LIN {X 0,Y 213.972,Z 422.456,A -85,B 0,C 180,E1 -20686.708,E2 -20686.708} C_VEL
LIN {X 0,Y 214.158,Z 422.425,A -85,B 0,C 180,E1 -20690.556,E2 -20690.556} C_VEL
LIN {X 0,Y 214.219,Z 422.426,A -85,B 0,C 180,E1 -20692.46,E2 -20692.46} C_VEL
LIN {X 0,Y 214.439,Z 422.398,A -85,B 0,C 180,E1 -20698.122,E2 -20698.122} C_VEL
LIN {X 0,Y 214.546,Z 422.38,A -85,B 0,C 180,E1 -20700,E2 -20700} C_VEL
LIN {X 0,Y 214.44,Z 422.395,A -85,B 0,C 180,E1 -20701.879,E2 -20701.879} C_VEL
LIN {X 0,Y 214.219,Z 422.4,A -85,B 0,C 180,E1 -20707.541,E2 -20707.541} C_VEL
LIN {X 0,Y 214.037,Z 422.432,A -85,B 0,C 180,E1 -20711.363,E2 -20711.363} C_VEL
LIN {X 0,Y 213.926,Z 422.461,A -85,B 0,C 180,E1 -20715.238,E2 -20715.238} C_VEL
LIN {X 0,Y 213.832,Z 422.475,A -85,B 0,C 180,E1 -20719.189,E2 -20719.189} C_VEL
LIN {X 0,Y 213.84,Z 422.469,A -85,B 0,C 180,E1 -20723.228,E2 -20723.228} C_VEL
LIN {X 0,Y 213.822,Z 422.463,A -85,B 0,C 180,E1 -20727.451,E2 -20727.451} C_VEL
LIN {X 0,Y 213.761,Z 422.467,A -85,B 0,C 180,E1 -20731.739,E2 -20731.739} C_VEL
LIN {X 0,Y 213.738,Z 422.473,A -85,B 0,C 180,E1 -20736.29,E2 -20736.29} C_VEL
LIN {X 0,Y 213.708,Z 422.488,A -85,B 0,C 180,E1 -20741.127,E2 -20741.127} C_VEL
LIN {X 0,Y 213.772,Z 422.468,A -85,B 0,C 180,E1 -20746.342,E2 -20746.342} C_VEL
LIN {X 0,Y 213.734,Z 422.475,A -85,B 0,C 180,E1 -20751.339,E2 -20751.339} C_VEL
LIN {X 0,Y 213.768,Z 422.481,A -85,B 0,C 180,E1 -20756.023,E2 -20756.023} C_VEL
LIN {X 0,Y 213.828,Z 422.466,A -85,B 0,C 180,E1 -20759.547,E2 -20759.547} C_VEL
LIN {X 0,Y 214.904,Z 425.409,A -85,B 0,C 180,E1 -20759.864,E2 -20759.864} C_VEL
LIN {X 0,Y 218.314,Z 431.493,A -85,B 0,C 180,E1 -20760.745,E2 -20760.745} C_VEL
LIN {X 0,Y 223.57,Z 442.478,A -85,B 0,C 180,E1 -20762.408,E2 -20762.408} C_VEL
LIN {X 0,Y 227.612,Z 453.444,A -85,B 0,C 180,E1 -20764.167,E2 -20764.167} C_VEL
LIN {X 0,Y 229.845,Z 460.684,A -85,B 0,C 180,E1 -20765.429,E2 -20765.429} C_VEL
LIN {X 0,Y 228.662,Z 469.845,A -85,B 0,C 180,E1 -20766.692,E2 -20766.692} C_VEL
LIN {X 0,Y 226.744,Z 480.14,A -85,B 0,C 180,E1 -20768.414,E2 -20768.414} C_VEL
LIN {X 0,Y 224.756,Z 489.465,A -85,B 0,C 180,E1 -20770.36,E2 -20770.36} C_VEL
LIN {X 0,Y 222.528,Z 498.031,A -85,B 0,C 180,E1 -20772.543,E2 -20772.543} C_VEL
LIN {X 0,Y 220.393,Z 506.343,A -85,B 0,C 180,E1 -20775.222,E2 -20775.222} C_VEL
LIN {X 0,Y 218.58,Z 512.97,A -85,B 0,C 180,E1 -20777.939,E2 -20777.939} C_VEL
LIN {X 0,Y 217.175,Z 518.259,A -85,B 0,C 180,E1 -20780.69,E2 -20780.69} C_VEL
LIN {X 0,Y 215.919,Z 522.415,A -85,B 0,C 180,E1 -20783.461,E2 -20783.461} C_VEL
LIN {X 0,Y 214.982,Z 525.535,A -85,B 0,C 180,E1 -20786.253,E2 -20786.253} C_VEL
LIN {X 0,Y 214.482,Z 528.213,A -85,B 0,C 180,E1 -20790.002,E2 -20790.002} C_VEL
LIN {X 0,Y 214.48,Z 528.919,A -85,B 0,C 180,E1 -20791.88,E2 -20791.88} C_VEL
LIN {X 0,Y 214.406,Z 529.283,A -85,B 0,C 180,E1 -20795.645,E2 -20795.645} C_VEL
LIN {X 0,Y 214.847,Z 528.85,A -85,B 0,C 180,E1 -20797.52,E2 -20797.52} C_VEL
LIN {X 0,Y 216.341,Z 526.738,A -85,B 0,C 180,E1 -20801.242,E2 -20801.242} C_VEL
LIN {X 0,Y 217.741,Z 523.653,A -85,B 0,C 180,E1 -20804.46,E2 -20804.46} C_VEL
LIN {X 0,Y 219.646,Z 519.074,A -85,B 0,C 180,E1 -20807.698,E2 -20807.698} C_VEL
LIN {X 0,Y 221.534,Z 513.949,A -85,B 0,C 180,E1 -20810.426,E2 -20810.426} C_VEL
LIN {X 0,Y 223.759,Z 507.49,A -85,B 0,C 180,E1 -20813.119,E2 -20813.119} C_VEL
LIN {X 0,Y 226.484,Z 499.387,A -85,B 0,C 180,E1 -20815.751,E2 -20815.751} C_VEL
LIN {X 0,Y 229.012,Z 490.992,A -85,B 0,C 180,E1 -20817.906,E2 -20817.906} C_VEL
LIN {X 0,Y 231.639,Z 480.659,A -85,B 0,C 180,E1 -20820.042,E2 -20820.042} C_VEL
LIN {X 0,Y 233.697,Z 470.671,A -85,B 0,C 180,E1 -20821.702,E2 -20821.702} C_VEL
LIN {X 0,Y 234.14,Z 467.189,A -85,B 0,C 180,E1 -20822.222,E2 -20822.222} C_VEL
LIN {X 0,Y 230.921,Z 456.648,A -85,B 0,C 180,E1 -20824.367,E2 -20824.367} C_VEL
LIN {X 0,Y 226.28,Z 445.434,A -85,B 0,C 180,E1 -20826.519,E2 -20826.519} C_VEL
LIN {X 0,Y 220.698,Z 434.511,A -85,B 0,C 180,E1 -20828.539,E2 -20828.539} C_VEL
LIN {X 0,Y 216.421,Z 427.342,A -85,B 0,C 180,E1 -20829.854,E2 -20829.854} C_VEL
LIN {X 0,Y 214.218,Z 424.278,A -85,B 0,C 180,E1 -20830.471,E2 -20830.471} C_VEL
LIN {X 0,Y 213.992,Z 423.665,A -85,B 0,C 180,E1 -20830.581,E2 -20830.581} C_VEL
LIN {X 0,Y 213.732,Z 422.486,A -85,B 0,C 180,E1 -20831.279,E2 -20831.279} C_VEL
LIN {X 0,Y 213.709,Z 422.483,A -85,B 0,C 180,E1 -20836.345,E2 -20836.345} C_VEL
LIN {X 0,Y 213.723,Z 422.461,A -85,B 0,C 180,E1 -20839.144,E2 -20839.144} C_VEL
LIN {X 0,Y 213.75,Z 422.463,A -85,B 0,C 180,E1 -20843.712,E2 -20843.712} C_VEL
LIN {X 0,Y 213.774,Z 422.437,A -85,B 0,C 180,E1 -20848.263,E2 -20848.263} C_VEL
LIN {X 0,Y 213.86,Z 422.536,A -85,B 0,C 180,E1 -20852.294,E2 -20852.294} C_VEL
LIN {X 0,Y 217.554,Z 436.442,A -85,B 0,C 180,E1 -20854.225,E2 -20854.225} C_VEL
LIN {X 0,Y 221.181,Z 450.157,A -85,B 0,C 180,E1 -20856.473,E2 -20856.473} C_VEL
LIN {X 0,Y 221.865,Z 453.454,A -85,B 0,C 180,E1 -20857.048,E2 -20857.048} C_VEL
LIN {X 0,Y 219.974,Z 466.735,A -85,B 0,C 180,E1 -20859.424,E2 -20859.424} C_VEL
LIN {X 0,Y 218.056,Z 479.392,A -85,B 0,C 180,E1 -20862.17,E2 -20862.17} C_VEL
LIN {X 0,Y 216.65,Z 490.066,A -85,B 0,C 180,E1 -20864.958,E2 -20864.958} C_VEL
LIN {X 0,Y 215.409,Z 500.374,A -85,B 0,C 180,E1 -20868.184,E2 -20868.184} C_VEL
LIN {X 0,Y 214.502,Z 509.16,A -85,B 0,C 180,E1 -20871.521,E2 -20871.521} C_VEL
LIN {X 0,Y 213.8,Z 517.298,A -85,B 0,C 180,E1 -20875.286,E2 -20875.286} C_VEL
LIN {X 0,Y 214.082,Z 523.832,A -85,B 0,C 180,E1 -20879.059,E2 -20879.059} C_VEL
LIN {X 0,Y 214.565,Z 528.917,A -85,B 0,C 180,E1 -20882.816,E2 -20882.816} C_VEL
LIN {X 0,Y 215.439,Z 531.828,A -85,B 0,C 180,E1 -20885.616,E2 -20885.616} C_VEL
LIN {X 0,Y 217.171,Z 534.69,A -85,B 0,C 180,E1 -20889.311,E2 -20889.311} C_VEL
LIN {X 0,Y 219.799,Z 536.336,A -85,B 0,C 180,E1 -20892.933,E2 -20892.933} C_VEL
LIN {X 0,Y 223.15,Z 536.823,A -85,B 0,C 180,E1 -20896.466,E2 -20896.466} C_VEL
LIN {X 0,Y 227.156,Z 536.219,A -85,B 0,C 180,E1 -20899.897,E2 -20899.897} C_VEL
LIN {X 0,Y 232.015,Z 534.486,A -85,B 0,C 180,E1 -20903.19,E2 -20903.19} C_VEL
LIN {X 0,Y 237.676,Z 531.614,A -85,B 0,C 180,E1 -20906.33,E2 -20906.33} C_VEL
LIN {X 0,Y 244.096,Z 527.588,A -85,B 0,C 180,E1 -20909.305,E2 -20909.305} C_VEL
LIN {X 0,Y 251.223,Z 522.349,A -85,B 0,C 180,E1 -20912.108,E2 -20912.108} C_VEL
LIN {X 0,Y 258.956,Z 515.86,A -85,B 0,C 180,E1 -20914.745,E2 -20914.745} C_VEL
LIN {X 0,Y 264.693,Z 510.488,A -85,B 0,C 180,E1 -20916.478,E2 -20916.478} C_VEL
LIN {X 0,Y 265.117,Z 509.97,A -85,B 0,C 180,E1 -20917.317,E2 -20917.317} C_VEL
LIN {X 0,Y 264.451,Z 510.646,A -85,B 0,C 180,E1 -20919.629,E2 -20919.629} C_VEL
LIN {X 0,Y 263.644,Z 512.309,A -85,B 0,C 180,E1 -20921.792,E2 -20921.792} C_VEL
LIN {X 0,Y 262.698,Z 513.804,A -85,B 0,C 180,E1 -20922.666,E2 -20922.666} C_VEL
LIN {X 0,Y 257.963,Z 521.137,A -85,B 0,C 180,E1 -20925.606,E2 -20925.606} C_VEL
LIN {X 0,Y 253.28,Z 528.754,A -85,B 0,C 180,E1 -20928.243,E2 -20928.243} C_VEL
LIN {X 0,Y 248.723,Z 535.889,A -85,B 0,C 180,E1 -20930.521,E2 -20930.521} C_VEL
LIN {X 0,Y 247.57,Z 537.606,A -85,B 0,C 180,E1 -20931.049,E2 -20931.049} C_VEL
LIN {X 0,Y 245.821,Z 539.886,A -85,B 0,C 180,E1 -20931.678,E2 -20931.678} C_VEL
LIN {X 0,Y 241.19,Z 544.542,A -85,B 0,C 180,E1 -20932.727,E2 -20932.727} C_VEL
LIN {X 0,Y 232.211,Z 552.188,A -85,B 0,C 180,E1 -20934.517,E2 -20934.517} C_VEL
LIN {X 0,Y 229.199,Z 555.116,A -85,B 0,C 180,E1 -20935.539,E2 -20935.539} C_VEL
LIN {X 0,Y 222.184,Z 562.638,A -85,B 0,C 180,E1 -20938.785,E2 -20938.785} C_VEL
LIN {X 0,Y 215.683,Z 569.927,A -85,B 0,C 180,E1 -20942.857,E2 -20942.857} C_VEL
LIN {X 0,Y 211.314,Z 574.923,A -85,B 0,C 180,E1 -20946.476,E2 -20946.476} C_VEL
LIN {X 0,Y 208.261,Z 578.95,A -85,B 0,C 180,E1 -20950.276,E2 -20950.276} C_VEL
LIN {X 0,Y 206.358,Z 581.976,A -85,B 0,C 180,E1 -20954.187,E2 -20954.187} C_VEL
LIN {X 0,Y 205.635,Z 584.262,A -85,B 0,C 180,E1 -20959.163,E2 -20959.163} C_VEL
LIN {X 0,Y 205.742,Z 586.841,A -85,B 0,C 180,E1 -20962.145,E2 -20962.145} C_VEL
LIN {X 0,Y 206.04,Z 588.139,A -85,B 0,C 180,E1 -20964.125,E2 -20964.125} C_VEL
LIN {X 0,Y 206.356,Z 588.982,A -85,B 0,C 180,E1 -20966.092,E2 -20966.092} C_VEL
LIN {X 0,Y 206.795,Z 589.425,A -85,B 0,C 180,E1 -20968.05,E2 -20968.05} C_VEL
LIN {X 0,Y 207.323,Z 589.463,A -85,B 0,C 180,E1 -20969.998,E2 -20969.998} C_VEL
LIN {X 0,Y 206.902,Z 588.899,A -85,B 0,C 180,E1 -20971.944,E2 -20971.944} C_VEL
LIN {X 0,Y 206.51,Z 587.894,A -85,B 0,C 180,E1 -20973.901,E2 -20973.901} C_VEL
LIN {X 0,Y 206.262,Z 586.479,A -85,B 0,C 180,E1 -20975.865,E2 -20975.865} C_VEL
LIN {X 0,Y 205.933,Z 584.151,A -85,B 0,C 180,E1 -20978.233,E2 -20978.233} C_VEL
LIN {X 0,Y 205.836,Z 579.365,A -85,B 0,C 180,E1 -20981.819,E2 -20981.819} C_VEL
LIN {X 0,Y 206.442,Z 573.1,A -85,B 0,C 180,E1 -20985.295,E2 -20985.295} C_VEL
LIN {X 0,Y 207.613,Z 565.906,A -85,B 0,C 180,E1 -20988.384,E2 -20988.384} C_VEL
LIN {X 0,Y 209.282,Z 557.808,A -85,B 0,C 180,E1 -20991.159,E2 -20991.159} C_VEL
LIN {X 0,Y 211.193,Z 549.183,A -85,B 0,C 180,E1 -20993.534,E2 -20993.534} C_VEL
LIN {X 0,Y 213.298,Z 538.785,A -85,B 0,C 180,E1 -20995.823,E2 -20995.823} C_VEL
LIN {X 0,Y 213.452,Z 527.585,A -85,B 0,C 180,E1 -20997.979,E2 -20997.979} C_VEL
LIN {X 0,Y 213.359,Z 515.663,A -85,B 0,C 180,E1 -20999.859,E2 -20999.859} C_VEL
LIN {X 0,Y 213.14,Z 502.394,A -85,B 0,C 180,E1 -21001.484,E2 -21001.484} C_VEL
LIN {X 0,Y 212.646,Z 488.731,A -85,B 0,C 180,E1 -21002.74,E2 -21002.74} C_VEL
LIN {X 0,Y 211.647,Z 474.631,A -85,B 0,C 180,E1 -21003.631,E2 -21003.631} C_VEL
LIN {X 0,Y 210.095,Z 466.817,A -85,B 0,C 180,E1 -21004.215,E2 -21004.215} C_VEL
LIN {X 0,Y 209.318,Z 453.606,A -85,B 0,C 180,E1 -21006.447,E2 -21006.447} C_VEL
LIN {X 0,Y 210.89,Z 446.822,A -85,B 0,C 180,E1 -21010.704,E2 -21010.704} C_VEL
LIN {X 0,Y 211.132,Z 445.184,A -85,B 0,C 180,E1 -21011.736,E2 -21011.736} C_VEL
LIN {X 0,Y 210.401,Z 440.852,A -85,B 0,C 180,E1 -21014.541,E2 -21014.541} C_VEL
LIN {X 0,Y 208.94,Z 434.226,A -85,B 0,C 180,E1 -21019.012,E2 -21019.012} C_VEL
LIN {X 0,Y 207.621,Z 427.738,A -85,B 0,C 180,E1 -21023.575,E2 -21023.575} C_VEL
LIN {X 0,Y 206.785,Z 423.349,A -85,B 0,C 180,E1 -21026.913,E2 -21026.913} C_VEL
LIN {X 0,Y 206.758,Z 423.354,A -85,B 0,C 180,E1 -21032.096,E2 -21032.096} C_VEL
LIN {X 0,Y 206.777,Z 423.351,A -85,B 0,C 180,E1 -21036.583,E2 -21036.583} C_VEL
LIN {X 0,Y 206.865,Z 423.341,A -85,B 0,C 180,E1 -21042.196,E2 -21042.196} C_VEL
LIN {X 0,Y 206.905,Z 423.334,A -85,B 0,C 180,E1 -21046.245,E2 -21046.245} C_VEL
LIN {X 0,Y 207.097,Z 423.303,A -85,B 0,C 180,E1 -21050.231,E2 -21050.231} C_VEL
LIN {X 0,Y 207.159,Z 423.304,A -85,B 0,C 180,E1 -21052.201,E2 -21052.201} C_VEL
LIN {X 0,Y 207.376,Z 423.278,A -85,B 0,C 180,E1 -21058.058,E2 -21058.058} C_VEL
LIN {X 0,Y 207.511,Z 423.256,A -85,B 0,C 180,E1 -21060,E2 -21060} C_VEL
LIN {X 0,Y 207.082,Z 423.315,A -85,B 0,C 180,E1 -21063.893,E2 -21063.893} C_VEL
LIN {X 0,Y 207.16,Z 423.275,A -85,B 0,C 180,E1 -21067.8,E2 -21067.8} C_VEL
LIN {X 0,Y 206.974,Z 423.316,A -85,B 0,C 180,E1 -21071.756,E2 -21071.756} C_VEL
LIN {X 0,Y 206.859,Z 423.34,A -85,B 0,C 180,E1 -21075.772,E2 -21075.772} C_VEL
LIN {X 0,Y 206.776,Z 423.353,A -85,B 0,C 180,E1 -21079.87,E2 -21079.87} C_VEL
LIN {X 0,Y 206.756,Z 423.354,A -85,B 0,C 180,E1 -21084.074,E2 -21084.074} C_VEL
LIN {X 0,Y 206.73,Z 423.331,A -85,B 0,C 180,E1 -21088.422,E2 -21088.422} C_VEL
LIN {X 0,Y 206.692,Z 423.358,A -85,B 0,C 180,E1 -21092.959,E2 -21092.959} C_VEL
LIN {X 0,Y 206.673,Z 423.341,A -85,B 0,C 180,E1 -21097.742,E2 -21097.742} C_VEL
LIN {X 0,Y 206.638,Z 423.369,A -85,B 0,C 180,E1 -21101.565,E2 -21101.565} C_VEL
LIN {X 0,Y 206.674,Z 423.347,A -85,B 0,C 180,E1 -21105.571,E2 -21105.571} C_VEL
LIN {X 0,Y 206.677,Z 423.358,A -85,B 0,C 180,E1 -21109.756,E2 -21109.756} C_VEL
LIN {X 0,Y 206.729,Z 423.358,A -85,B 0,C 180,E1 -21114.698,E2 -21114.698} C_VEL
LIN {X 0,Y 206.75,Z 423.408,A -85,B 0,C 180,E1 -21118.315,E2 -21118.315} C_VEL
LIN {X 0,Y 207.722,Z 426.15,A -85,B 0,C 180,E1 -21118.613,E2 -21118.613} C_VEL
LIN {X 0,Y 209.214,Z 428.525,A -85,B 0,C 180,E1 -21119.003,E2 -21119.003} C_VEL
LIN {X 0,Y 214.487,Z 438.615,A -85,B 0,C 180,E1 -21120.587,E2 -21120.587} C_VEL
LIN {X 0,Y 218.44,Z 447.417,A -85,B 0,C 180,E1 -21122.047,E2 -21122.047} C_VEL
LIN {X 0,Y 222.032,Z 457.851,A -85,B 0,C 180,E1 -21123.866,E2 -21123.866} C_VEL
LIN {X 0,Y 223.515,Z 463.341,A -85,B 0,C 180,E1 -21124.882,E2 -21124.882} C_VEL
LIN {X 0,Y 221.521,Z 475.252,A -85,B 0,C 180,E1 -21126.638,E2 -21126.638} C_VEL
LIN {X 0,Y 219.438,Z 485.12,A -85,B 0,C 180,E1 -21128.489,E2 -21128.489} C_VEL
LIN {X 0,Y 217.232,Z 494.292,A -85,B 0,C 180,E1 -21130.636,E2 -21130.636} C_VEL
LIN {X 0,Y 215.061,Z 502.163,A -85,B 0,C 180,E1 -21132.898,E2 -21132.898} C_VEL
LIN {X 0,Y 212.983,Z 509.845,A -85,B 0,C 180,E1 -21135.674,E2 -21135.674} C_VEL
LIN {X 0,Y 211.137,Z 516.01,A -85,B 0,C 180,E1 -21138.482,E2 -21138.482} C_VEL
LIN {X 0,Y 209.81,Z 520.862,A -85,B 0,C 180,E1 -21141.333,E2 -21141.333} C_VEL
LIN {X 0,Y 208.557,Z 524.649,A -85,B 0,C 180,E1 -21144.2,E2 -21144.2} C_VEL
LIN {X 0,Y 207.612,Z 528.119,A -85,B 0,C 180,E1 -21148.062,E2 -21148.062} C_VEL
LIN {X 0,Y 207.455,Z 529.242,A -85,B 0,C 180,E1 -21150.002,E2 -21150.002} C_VEL
LIN {X 0,Y 207.456,Z 529.937,A -85,B 0,C 180,E1 -21151.943,E2 -21151.943} C_VEL
LIN {X 0,Y 207.407,Z 530.284,A -85,B 0,C 180,E1 -21155.837,E2 -21155.837} C_VEL
LIN {X 0,Y 207.875,Z 529.832,A -85,B 0,C 180,E1 -21157.774,E2 -21157.774} C_VEL
LIN {X 0,Y 209.449,Z 527.701,A -85,B 0,C 180,E1 -21161.617,E2 -21161.617} C_VEL
LIN {X 0,Y 210.931,Z 524.609,A -85,B 0,C 180,E1 -21164.925,E2 -21164.925} C_VEL
LIN {X 0,Y 212.953,Z 519.986,A -85,B 0,C 180,E1 -21168.274,E2 -21168.274} C_VEL
LIN {X 0,Y 214.942,Z 514.84,A -85,B 0,C 180,E1 -21171.082,E2 -21171.082} C_VEL
LIN {X 0,Y 217.3,Z 508.353,A -85,B 0,C 180,E1 -21173.848,E2 -21173.848} C_VEL
LIN {X 0,Y 220.157,Z 500.205,A -85,B 0,C 180,E1 -21176.548,E2 -21176.548} C_VEL
LIN {X 0,Y 222.803,Z 491.771,A -85,B 0,C 180,E1 -21178.755,E2 -21178.755} C_VEL
LIN {X 0,Y 225.555,Z 481.392,A -85,B 0,C 180,E1 -21180.94,E2 -21180.94} C_VEL
LIN {X 0,Y 227.729,Z 471.327,A -85,B 0,C 180,E1 -21182.634,E2 -21182.634} C_VEL
LIN {X 0,Y 227.957,Z 470.157,A -85,B 0,C 180,E1 -21182.8,E2 -21182.8} C_VEL
LIN {X 0,Y 225.533,Z 461.174,A -85,B 0,C 180,E1 -21184.727,E2 -21184.727} C_VEL
LIN {X 0,Y 221.594,Z 450.819,A -85,B 0,C 180,E1 -21186.867,E2 -21186.867} C_VEL
LIN {X 0,Y 216.859,Z 441.027,A -85,B 0,C 180,E1 -21188.847,E2 -21188.847} C_VEL
LIN {X 0,Y 211.559,Z 431.787,A -85,B 0,C 180,E1 -21190.696,E2 -21190.696} C_VEL
LIN {X 0,Y 208.535,Z 427.317,A -85,B 0,C 180,E1 -21191.643,E2 -21191.643} C_VEL
LIN {X 0,Y 206.975,Z 424.661,A -85,B 0,C 180,E1 -21192.211,E2 -21192.211} C_VEL
LIN {X 0,Y 206.67,Z 423.361,A -85,B 0,C 180,E1 -21193.01,E2 -21193.01} C_VEL
LIN {X 0,Y 206.629,Z 423.372,A -85,B 0,C 180,E1 -21197.136,E2 -21197.136} C_VEL
LIN {X 0,Y 206.693,Z 423.318,A -85,B 0,C 180,E1 -21201.451,E2 -21201.451} C_VEL
LIN {X 0,Y 206.706,Z 423.358,A -85,B 0,C 180,E1 -21204.689,E2 -21204.689} C_VEL
LIN {X 0,Y 206.716,Z 423.302,A -85,B 0,C 180,E1 -21209.337,E2 -21209.337} C_VEL
LIN {X 0,Y 206.791,Z 423.297,A -85,B 0,C 180,E1 -21211.89,E2 -21211.89} C_VEL
LIN {X 0,Y 210.85,Z 438.804,A -85,B 0,C 180,E1 -21214.156,E2 -21214.156} C_VEL
LIN {X 0,Y 214.533,Z 452.675,A -85,B 0,C 180,E1 -21216.533,E2 -21216.533} C_VEL
LIN {X 0,Y 214.763,Z 454.641,A -85,B 0,C 180,E1 -21216.877,E2 -21216.877} C_VEL
LIN {X 0,Y 212.671,Z 468.408,A -85,B 0,C 180,E1 -21219.444,E2 -21219.444} C_VEL
LIN {X 0,Y 210.976,Z 480.013,A -85,B 0,C 180,E1 -21222.053,E2 -21222.053} C_VEL
LIN {X 0,Y 209.519,Z 490.722,A -85,B 0,C 180,E1 -21224.932,E2 -21224.932} C_VEL
LIN {X 0,Y 208.221,Z 501.251,A -85,B 0,C 180,E1 -21228.315,E2 -21228.315} C_VEL
LIN {X 0,Y 207.348,Z 509.968,A -85,B 0,C 180,E1 -21231.717,E2 -21231.717} C_VEL
LIN {X 0,Y 206.729,Z 517.255,A -85,B 0,C 180,E1 -21235.124,E2 -21235.124} C_VEL
LIN {X 0,Y 207.002,Z 524.028,A -85,B 0,C 180,E1 -21239.027,E2 -21239.027} C_VEL
LIN {X 0,Y 207.512,Z 529.372,A -85,B 0,C 180,E1 -21242.912,E2 -21242.912} C_VEL
LIN {X 0,Y 208.407,Z 532.537,A -85,B 0,C 180,E1 -21245.806,E2 -21245.806} C_VEL
LIN {X 0,Y 210.254,Z 535.659,A -85,B 0,C 180,E1 -21249.621,E2 -21249.621} C_VEL
LIN {X 0,Y 213.011,Z 537.583,A -85,B 0,C 180,E1 -21253.353,E2 -21253.353} C_VEL
LIN {X 0,Y 216.518,Z 538.362,A -85,B 0,C 180,E1 -21256.985,E2 -21256.985} C_VEL
LIN {X 0,Y 220.722,Z 538.064,A -85,B 0,C 180,E1 -21260.502,E2 -21260.502} C_VEL
LIN {X 0,Y 225.829,Z 536.652,A -85,B 0,C 180,E1 -21263.864,E2 -21263.864} C_VEL
LIN {X 0,Y 231.735,Z 534.129,A -85,B 0,C 180,E1 -21267.059,E2 -21267.059} C_VEL
LIN {X 0,Y 238.438,Z 530.473,A -85,B 0,C 180,E1 -21270.071,E2 -21270.071} C_VEL
LIN {X 0,Y 245.837,Z 525.649,A -85,B 0,C 180,E1 -21272.9,E2 -21272.9} C_VEL
LIN {X 0,Y 253.858,Z 519.627,A -85,B 0,C 180,E1 -21275.547,E2 -21275.547} C_VEL
LIN {X 0,Y 259.777,Z 514.726,A -85,B 0,C 180,E1 -21277.355,E2 -21277.355} C_VEL
LIN {X 0,Y 259.438,Z 515.056,A -85,B 0,C 180,E1 -21278.539,E2 -21278.539} C_VEL
LIN {X 0,Y 258.737,Z 516.294,A -85,B 0,C 180,E1 -21280.685,E2 -21280.685} C_VEL
LIN {X 0,Y 258.233,Z 517.213,A -85,B 0,C 180,E1 -21281.58,E2 -21281.58} C_VEL
LIN {X 0,Y 255.122,Z 521.41,A -85,B 0,C 180,E1 -21283.526,E2 -21283.526} C_VEL
LIN {X 0,Y 250.58,Z 527.832,A -85,B 0,C 180,E1 -21286.038,E2 -21286.038} C_VEL
LIN {X 0,Y 245.146,Z 535.558,A -85,B 0,C 180,E1 -21288.746,E2 -21288.746} C_VEL
LIN {X 0,Y 239.114,Z 543.422,A -85,B 0,C 180,E1 -21291.347,E2 -21291.347} C_VEL
LIN {X 0,Y 230.97,Z 552.989,A -85,B 0,C 180,E1 -21294.679,E2 -21294.679} C_VEL
LIN {X 0,Y 229.199,Z 555.116,A -85,B 0,C 180,E1 -21295.539,E2 -21295.539} C_VEL
LIN {X 0,Y 226.963,Z 557.085,A -85,B 0,C 180,E1 -21296.213,E2 -21296.213} C_VEL
LIN {X 0,Y 221.842,Z 560.15,A -85,B 0,C 180,E1 -21297.043,E2 -21297.043} C_VEL
LIN {X 0,Y 216.728,Z 562.955,A -85,B 0,C 180,E1 -21297.932,E2 -21297.932} C_VEL
LIN {X 0,Y 214.536,Z 564.539,A -85,B 0,C 180,E1 -21298.698,E2 -21298.698} C_VEL
LIN {X 0,Y 208.094,Z 571.002,A -85,B 0,C 180,E1 -21302.873,E2 -21302.873} C_VEL
LIN {X 0,Y 204.748,Z 574.437,A -85,B 0,C 180,E1 -21305.674,E2 -21305.674} C_VEL
LIN {X 0,Y 201.52,Z 578.132,A -85,B 0,C 180,E1 -21309.587,E2 -21309.587} C_VEL
LIN {X 0,Y 199.477,Z 580.864,A -85,B 0,C 180,E1 -21313.627,E2 -21313.627} C_VEL
LIN {X 0,Y 198.616,Z 583.13,A -85,B 0,C 180,E1 -21318.776,E2 -21318.776} C_VEL
LIN {X 0,Y 198.668,Z 586.03,A -85,B 0,C 180,E1 -21322.102,E2 -21322.102} C_VEL
LIN {X 0,Y 198.93,Z 587.137,A -85,B 0,C 180,E1 -21323.914,E2 -21323.914} C_VEL
LIN {X 0,Y 199.284,Z 587.981,A -85,B 0,C 180,E1 -21325.953,E2 -21325.953} C_VEL
LIN {X 0,Y 199.719,Z 588.417,A -85,B 0,C 180,E1 -21327.981,E2 -21327.981} C_VEL
LIN {X 0,Y 200.279,Z 588.451,A -85,B 0,C 180,E1 -21329.998,E2 -21329.998} C_VEL
LIN {X 0,Y 199.826,Z 587.868,A -85,B 0,C 180,E1 -21332.013,E2 -21332.013} C_VEL
LIN {X 0,Y 199.438,Z 586.853,A -85,B 0,C 180,E1 -21334.039,E2 -21334.039} C_VEL
LIN {X 0,Y 199.164,Z 585.424,A -85,B 0,C 180,E1 -21336.075,E2 -21336.075} C_VEL
LIN {X 0,Y 198.809,Z 582.499,A -85,B 0,C 180,E1 -21339.048,E2 -21339.048} C_VEL
LIN {X 0,Y 198.803,Z 578.268,A -85,B 0,C 180,E1 -21342.244,E2 -21342.244} C_VEL
LIN {X 0,Y 199.515,Z 571.976,A -85,B 0,C 180,E1 -21345.84,E2 -21345.84} C_VEL
LIN {X 0,Y 200.883,Z 564.435,A -85,B 0,C 180,E1 -21349.16,E2 -21349.16} C_VEL
LIN {X 0,Y 202.6,Z 556.64,A -85,B 0,C 180,E1 -21351.892,E2 -21351.892} C_VEL
LIN {X 0,Y 204.571,Z 547.963,A -85,B 0,C 180,E1 -21354.344,E2 -21354.344} C_VEL
LIN {X 0,Y 206.455,Z 539.639,A -85,B 0,C 180,E1 -21356.263,E2 -21356.263} C_VEL
LIN {X 0,Y 206.742,Z 527.701,A -85,B 0,C 180,E1 -21358.693,E2 -21358.693} C_VEL
LIN {X 0,Y 206.828,Z 515.981,A -85,B 0,C 180,E1 -21360.641,E2 -21360.641} C_VEL
LIN {X 0,Y 206.765,Z 503.366,A -85,B 0,C 180,E1 -21362.296,E2 -21362.296} C_VEL
LIN {X 0,Y 206.443,Z 489.769,A -85,B 0,C 180,E1 -21363.635,E2 -21363.635} C_VEL
LIN {X 0,Y 205.65,Z 476.251,A -85,B 0,C 180,E1 -21364.585,E2 -21364.585} C_VEL
LIN {X 0,Y 203.515,Z 465.411,A -85,B 0,C 180,E1 -21365.47,E2 -21365.47} C_VEL
LIN {X 0,Y 202.742,Z 451.207,A -85,B 0,C 180,E1 -21368.021,E2 -21368.021} C_VEL
LIN {X 0,Y 203.835,Z 446.764,A -85,B 0,C 180,E1 -21370.924,E2 -21370.924} C_VEL
LIN {X 0,Y 203.855,Z 443.815,A -85,B 0,C 180,E1 -21372.878,E2 -21372.878} C_VEL
LIN {X 0,Y 202.274,Z 436.796,A -85,B 0,C 180,E1 -21377.698,E2 -21377.698} C_VEL
LIN {X 0,Y 200.965,Z 430.427,A -85,B 0,C 180,E1 -21382.266,E2 -21382.266} C_VEL
LIN {X 0,Y 199.742,Z 424.226,A -85,B 0,C 180,E1 -21387.045,E2 -21387.045} C_VEL
LIN {X 0,Y 199.704,Z 424.23,A -85,B 0,C 180,E1 -21391.612,E2 -21391.612} C_VEL
LIN {X 0,Y 199.73,Z 424.233,A -85,B 0,C 180,E1 -21397.229,E2 -21397.229} C_VEL
LIN {X 0,Y 199.788,Z 424.223,A -85,B 0,C 180,E1 -21401.757,E2 -21401.757} C_VEL
LIN {X 0,Y 199.84,Z 424.213,A -85,B 0,C 180,E1 -21405.749,E2 -21405.749} C_VEL
LIN {X 0,Y 200.061,Z 424.179,A -85,B 0,C 180,E1 -21409.884,E2 -21409.884} C_VEL
LIN {X 0,Y 200.027,Z 424.191,A -85,B 0,C 180,E1 -21413.95,E2 -21413.95} C_VEL
LIN {X 0,Y 200.315,Z 424.158,A -85,B 0,C 180,E1 -21417.99,E2 -21417.99} C_VEL
LIN {X 0,Y 200.475,Z 424.132,A -85,B 0,C 180,E1 -21420.001,E2 -21420.001} C_VEL
LIN {X 0,Y 200.027,Z 424.194,A -85,B 0,C 180,E1 -21424.03,E2 -21424.03} C_VEL
LIN {X 0,Y 200.103,Z 424.15,A -85,B 0,C 180,E1 -21428.077,E2 -21428.077} C_VEL
LIN {X 0,Y 199.906,Z 424.2,A -85,B 0,C 180,E1 -21432.178,E2 -21432.178} C_VEL
LIN {X 0,Y 199.797,Z 424.217,A -85,B 0,C 180,E1 -21436.345,E2 -21436.345} C_VEL
LIN {X 0,Y 199.692,Z 424.234,A -85,B 0,C 180,E1 -21440.607,E2 -21440.607} C_VEL
LIN {X 0,Y 199.666,Z 424.239,A -85,B 0,C 180,E1 -21444.986,E2 -21444.986} C_VEL
LIN {X 0,Y 199.658,Z 424.204,A -85,B 0,C 180,E1 -21449.526,E2 -21449.526} C_VEL
LIN {X 0,Y 199.665,Z 424.228,A -85,B 0,C 180,E1 -21452.357,E2 -21452.357} C_VEL
LIN {X 0,Y 199.617,Z 424.226,A -85,B 0,C 180,E1 -21456.765,E2 -21456.765} C_VEL
LIN {X 0,Y 199.602,Z 424.224,A -85,B 0,C 180,E1 -21459.33,E2 -21459.33} C_VEL
LIN {X 0,Y 199.571,Z 424.251,A -85,B 0,C 180,E1 -21462.313,E2 -21462.313} C_VEL
LIN {X 0,Y 199.608,Z 424.226,A -85,B 0,C 180,E1 -21465.24,E2 -21465.24} C_VEL
LIN {X 0,Y 199.62,Z 424.245,A -85,B 0,C 180,E1 -21468.019,E2 -21468.019} C_VEL
LIN {X 0,Y 199.64,Z 424.229,A -85,B 0,C 180,E1 -21470.759,E2 -21470.759} C_VEL
LIN {X 0,Y 199.633,Z 424.242,A -85,B 0,C 180,E1 -21475.721,E2 -21475.721} C_VEL
LIN {X 0,Y 199.657,Z 424.238,A -85,B 0,C 180,E1 -21476.929,E2 -21476.929} C_VEL
LIN {X 0,Y 200.767,Z 427.243,A -85,B 0,C 180,E1 -21477.314,E2 -21477.314} C_VEL
LIN {X 0,Y 202.14,Z 429.261,A -85,B 0,C 180,E1 -21477.688,E2 -21477.688} C_VEL
LIN {X 0,Y 207.837,Z 439.862,A -85,B 0,C 180,E1 -21479.492,E2 -21479.492} C_VEL
LIN {X 0,Y 212.571,Z 450.642,A -85,B 0,C 180,E1 -21481.405,E2 -21481.405} C_VEL
LIN {X 0,Y 216.133,Z 461.37,A -85,B 0,C 180,E1 -21483.408,E2 -21483.408} C_VEL
LIN {X 0,Y 217.102,Z 464.948,A -85,B 0,C 180,E1 -21484.12,E2 -21484.12} C_VEL
LIN {X 0,Y 215.136,Z 476.543,A -85,B 0,C 180,E1 -21485.902,E2 -21485.902} C_VEL
LIN {X 0,Y 212.956,Z 486.347,A -85,B 0,C 180,E1 -21487.8,E2 -21487.8} C_VEL
LIN {X 0,Y 210.637,Z 495.486,A -85,B 0,C 180,E1 -21490.004,E2 -21490.004} C_VEL
LIN {X 0,Y 208.377,Z 503.326,A -85,B 0,C 180,E1 -21492.332,E2 -21492.332} C_VEL
LIN {X 0,Y 206.195,Z 510.983,A -85,B 0,C 180,E1 -21495.191,E2 -21495.191} C_VEL
LIN {X 0,Y 204.271,Z 517.112,A -85,B 0,C 180,E1 -21498.089,E2 -21498.089} C_VEL
LIN {X 0,Y 202.872,Z 521.944,A -85,B 0,C 180,E1 -21501.034,E2 -21501.034} C_VEL
LIN {X 0,Y 201.57,Z 525.711,A -85,B 0,C 180,E1 -21503.998,E2 -21503.998} C_VEL
LIN {X 0,Y 200.591,Z 529.164,A -85,B 0,C 180,E1 -21507.994,E2 -21507.994} C_VEL
LIN {X 0,Y 200.428,Z 530.27,A -85,B 0,C 180,E1 -21510.002,E2 -21510.002} C_VEL
LIN {X 0,Y 200.431,Z 530.954,A -85,B 0,C 180,E1 -21512.012,E2 -21512.012} C_VEL
LIN {X 0,Y 200.41,Z 531.284,A -85,B 0,C 180,E1 -21516.041,E2 -21516.041} C_VEL
LIN {X 0,Y 200.908,Z 530.814,A -85,B 0,C 180,E1 -21518.046,E2 -21518.046} C_VEL
LIN {X 0,Y 202.567,Z 528.664,A -85,B 0,C 180,E1 -21522.017,E2 -21522.017} C_VEL
LIN {X 0,Y 204.143,Z 525.555,A -85,B 0,C 180,E1 -21525.429,E2 -21525.429} C_VEL
LIN {X 0,Y 206.278,Z 520.9,A -85,B 0,C 180,E1 -21528.887,E2 -21528.887} C_VEL
LIN {X 0,Y 208.756,Z 514.766,A -85,B 0,C 180,E1 -21532.258,E2 -21532.258} C_VEL
LIN {X 0,Y 211.366,Z 507.983,A -85,B 0,C 180,E1 -21535.086,E2 -21535.086} C_VEL
LIN {X 0,Y 214.368,Z 499.605,A -85,B 0,C 180,E1 -21537.8,E2 -21537.8} C_VEL
LIN {X 0,Y 217.184,Z 490.669,A -85,B 0,C 180,E1 -21540.106,E2 -21540.106} C_VEL
LIN {X 0,Y 219.804,Z 480.936,A -85,B 0,C 180,E1 -21542.113,E2 -21542.113} C_VEL
LIN {X 0,Y 221.788,Z 471.974,A -85,B 0,C 180,E1 -21543.622,E2 -21543.622} C_VEL
LIN {X 0,Y 219.147,Z 462.805,A -85,B 0,C 180,E1 -21545.738,E2 -21545.738} C_VEL
LIN {X 0,Y 215.415,Z 452.841,A -85,B 0,C 180,E1 -21547.919,E2 -21547.919} C_VEL
LIN {X 0,Y 210.649,Z 442.895,A -85,B 0,C 180,E1 -21550.067,E2 -21550.067} C_VEL
LIN {X 0,Y 204.762,Z 432.903,A -85,B 0,C 180,E1 -21552.26,E2 -21552.26} C_VEL
LIN {X 0,Y 201.17,Z 427.826,A -85,B 0,C 180,E1 -21553.463,E2 -21553.463} C_VEL
LIN {X 0,Y 200.051,Z 425.932,A -85,B 0,C 180,E1 -21553.943,E2 -21553.943} C_VEL
LIN {X 0,Y 199.601,Z 424.24,A -85,B 0,C 180,E1 -21555.013,E2 -21555.013} C_VEL
LIN {X 0,Y 199.585,Z 424.243,A -85,B 0,C 180,E1 -21558.005,E2 -21558.005} C_VEL
LIN {X 0,Y 199.615,Z 424.2,A -85,B 0,C 180,E1 -21560.769,E2 -21560.769} C_VEL
LIN {X 0,Y 199.62,Z 424.246,A -85,B 0,C 180,E1 -21565.714,E2 -21565.714} C_VEL
LIN {X 0,Y 199.699,Z 424.189,A -85,B 0,C 180,E1 -21568.136,E2 -21568.136} C_VEL
LIN {X 0,Y 199.721,Z 424.173,A -85,B 0,C 180,E1 -21571.523,E2 -21571.523} C_VEL
LIN {X 0,Y 203.678,Z 439.269,A -85,B 0,C 180,E1 -21573.788,E2 -21573.788} C_VEL
LIN {X 0,Y 207.343,Z 453.171,A -85,B 0,C 180,E1 -21576.235,E2 -21576.235} C_VEL
LIN {X 0,Y 207.657,Z 455.795,A -85,B 0,C 180,E1 -21576.711,E2 -21576.711} C_VEL
LIN {X 0,Y 205.602,Z 468.864,A -85,B 0,C 180,E1 -21579.228,E2 -21579.228} C_VEL
LIN {X 0,Y 203.878,Z 480.515,A -85,B 0,C 180,E1 -21581.925,E2 -21581.925} C_VEL
LIN {X 0,Y 202.389,Z 491.306,A -85,B 0,C 180,E1 -21584.903,E2 -21584.903} C_VEL
LIN {X 0,Y 201.257,Z 500.479,A -85,B 0,C 180,E1 -21587.905,E2 -21587.905} C_VEL
LIN {X 0,Y 200.322,Z 509.545,A -85,B 0,C 180,E1 -21591.424,E2 -21591.424} C_VEL
LIN {X 0,Y 199.662,Z 517.102,A -85,B 0,C 180,E1 -21594.951,E2 -21594.951} C_VEL
LIN {X 0,Y 199.924,Z 524.189,A -85,B 0,C 180,E1 -21598.992,E2 -21598.992} C_VEL
LIN {X 0,Y 200.436,Z 529.793,A -85,B 0,C 180,E1 -21603.014,E2 -21603.014} C_VEL
LIN {X 0,Y 201.369,Z 533.141,A -85,B 0,C 180,E1 -21606.01,E2 -21606.01} C_VEL
LIN {X 0,Y 203.319,Z 536.541,A -85,B 0,C 180,E1 -21609.952,E2 -21609.952} C_VEL
LIN {X 0,Y 206.202,Z 538.752,A -85,B 0,C 180,E1 -21613.802,E2 -21613.802} C_VEL
LIN {X 0,Y 209.896,Z 539.822,A -85,B 0,C 180,E1 -21617.538,E2 -21617.538} C_VEL
LIN {X 0,Y 214.298,Z 539.828,A -85,B 0,C 180,E1 -21621.146,E2 -21621.146} C_VEL
LIN {X 0,Y 219.646,Z 538.739,A -85,B 0,C 180,E1 -21624.579,E2 -21624.579} C_VEL
LIN {X 0,Y 225.816,Z 536.57,A -85,B 0,C 180,E1 -21627.829,E2 -21627.829} C_VEL
LIN {X 0,Y 234.653,Z 532.328,A -85,B 0,C 180,E1 -21631.61,E2 -21631.61} C_VEL
LIN {X 0,Y 242.518,Z 527.635,A -85,B 0,C 180,E1 -21634.409,E2 -21634.409} C_VEL
LIN {X 0,Y 250.99,Z 521.787,A -85,B 0,C 180,E1 -21637.015,E2 -21637.015} C_VEL
LIN {X 0,Y 253.191,Z 520.157,A -85,B 0,C 180,E1 -21637.638,E2 -21637.638} C_VEL
LIN {X 0,Y 253.749,Z 519.999,A -85,B 0,C 180,E1 -21639.147,E2 -21639.147} C_VEL
LIN {X 0,Y 252.559,Z 521.908,A -85,B 0,C 180,E1 -21641.292,E2 -21641.292} C_VEL
LIN {X 0,Y 247.902,Z 527.621,A -85,B 0,C 180,E1 -21643.878,E2 -21643.878} C_VEL
LIN {X 0,Y 243.06,Z 533.771,A -85,B 0,C 180,E1 -21646.291,E2 -21646.291} C_VEL
LIN {X 0,Y 236.527,Z 541.712,A -85,B 0,C 180,E1 -21649.178,E2 -21649.178} C_VEL
LIN {X 0,Y 230.778,Z 547.984,A -85,B 0,C 180,E1 -21651.367,E2 -21651.367} C_VEL
LIN {X 0,Y 221.874,Z 557.492,A -85,B 0,C 180,E1 -21655.237,E2 -21655.237} C_VEL
LIN {X 0,Y 215.828,Z 563.241,A -85,B 0,C 180,E1 -21657.979,E2 -21657.979} C_VEL
LIN {X 0,Y 214.536,Z 564.539,A -85,B 0,C 180,E1 -21658.698,E2 -21658.698} C_VEL
LIN {X 0,Y 211.674,Z 566.832,A -85,B 0,C 180,E1 -21659.952,E2 -21659.952} C_VEL
LIN {X 0,Y 205.565,Z 570.191,A -85,B 0,C 180,E1 -21661.903,E2 -21661.903} C_VEL
LIN {X 0,Y 199.807,Z 573.004,A -85,B 0,C 180,E1 -21664.03,E2 -21664.03} C_VEL
LIN {X 0,Y 197.551,Z 574.483,A -85,B 0,C 180,E1 -21665.533,E2 -21665.533} C_VEL
LIN {X 0,Y 193.54,Z 578.623,A -85,B 0,C 180,E1 -21670.922,E2 -21670.922} C_VEL
LIN {X 0,Y 192.042,Z 580.616,A -85,B 0,C 180,E1 -21675.155,E2 -21675.155} C_VEL
LIN {X 0,Y 191.645,Z 581.584,A -85,B 0,C 180,E1 -21677.825,E2 -21677.825} C_VEL
LIN {X 0,Y 191.605,Z 585.174,A -85,B 0,C 180,E1 -21682.032,E2 -21682.032} C_VEL
LIN {X 0,Y 192.209,Z 586.979,A -85,B 0,C 180,E1 -21685.804,E2 -21685.804} C_VEL
LIN {X 0,Y 192.643,Z 587.409,A -85,B 0,C 180,E1 -21687.907,E2 -21687.907} C_VEL
LIN {X 0,Y 193.233,Z 587.438,A -85,B 0,C 180,E1 -21689.998,E2 -21689.998} C_VEL
LIN {X 0,Y 192.749,Z 586.836,A -85,B 0,C 180,E1 -21692.087,E2 -21692.087} C_VEL
LIN {X 0,Y 192.365,Z 585.813,A -85,B 0,C 180,E1 -21694.188,E2 -21694.188} C_VEL
LIN {X 0,Y 192.049,Z 584.366,A -85,B 0,C 180,E1 -21696.301,E2 -21696.301} C_VEL
LIN {X 0,Y 191.708,Z 581.305,A -85,B 0,C 180,E1 -21699.493,E2 -21699.493} C_VEL
LIN {X 0,Y 191.756,Z 577.167,A -85,B 0,C 180,E1 -21702.701,E2 -21702.701} C_VEL
LIN {X 0,Y 192.573,Z 570.844,A -85,B 0,C 180,E1 -21706.427,E2 -21706.427} C_VEL
LIN {X 0,Y 193.916,Z 564.016,A -85,B 0,C 180,E1 -21709.559,E2 -21709.559} C_VEL
LIN {X 0,Y 195.943,Z 555.468,A -85,B 0,C 180,E1 -21712.677,E2 -21712.677} C_VEL
LIN {X 0,Y 198.025,Z 546.745,A -85,B 0,C 180,E1 -21715.204,E2 -21715.204} C_VEL
LIN {X 0,Y 199.631,Z 539.479,A -85,B 0,C 180,E1 -21716.951,E2 -21716.951} C_VEL
LIN {X 0,Y 200.014,Z 529.542,A -85,B 0,C 180,E1 -21719.123,E2 -21719.123} C_VEL
LIN {X 0,Y 200.24,Z 518.206,A -85,B 0,C 180,E1 -21721.175,E2 -21721.175} C_VEL
LIN {X 0,Y 200.436,Z 505.745,A -85,B 0,C 180,E1 -21722.962,E2 -21722.962} C_VEL
LIN {X 0,Y 200.334,Z 492.335,A -85,B 0,C 180,E1 -21724.447,E2 -21724.447} C_VEL
LIN {X 0,Y 199.865,Z 479.051,A -85,B 0,C 180,E1 -21725.485,E2 -21725.485} C_VEL
LIN {X 0,Y 197.112,Z 464.705,A -85,B 0,C 180,E1 -21726.702,E2 -21726.702} C_VEL
LIN {X 0,Y 196.461,Z 452.98,A -85,B 0,C 180,E1 -21728.916,E2 -21728.916} C_VEL
LIN {X 0,Y 196.274,Z 448.67,A -85,B 0,C 180,E1 -21729.792,E2 -21729.792} C_VEL
LIN {X 0,Y 196.779,Z 446.289,A -85,B 0,C 180,E1 -21731.408,E2 -21731.408} C_VEL
LIN {X 0,Y 196.561,Z 443.263,A -85,B 0,C 180,E1 -21733.507,E2 -21733.507} C_VEL
LIN {X 0,Y 195.055,Z 436.727,A -85,B 0,C 180,E1 -21738.187,E2 -21738.187} C_VEL
LIN {X 0,Y 193.705,Z 430.348,A -85,B 0,C 180,E1 -21742.954,E2 -21742.954} C_VEL
LIN {X 0,Y 192.716,Z 425.101,A -85,B 0,C 180,E1 -21747.113,E2 -21747.113} C_VEL
LIN {X 0,Y 192.657,Z 425.108,A -85,B 0,C 180,E1 -21751.691,E2 -21751.691} C_VEL
LIN {X 0,Y 192.697,Z 425.104,A -85,B 0,C 180,E1 -21756.348,E2 -21756.348} C_VEL
LIN {X 0,Y 192.723,Z 425.103,A -85,B 0,C 180,E1 -21761.457,E2 -21761.457} C_VEL
LIN {X 0,Y 192.765,Z 425.091,A -85,B 0,C 180,E1 -21765.214,E2 -21765.214} C_VEL
LIN {X 0,Y 192.972,Z 425.063,A -85,B 0,C 180,E1 -21769.508,E2 -21769.508} C_VEL
LIN {X 0,Y 193.053,Z 425.062,A -85,B 0,C 180,E1 -21771.627,E2 -21771.627} C_VEL
LIN {X 0,Y 193.257,Z 425.037,A -85,B 0,C 180,E1 -21777.916,E2 -21777.916} C_VEL
LIN {X 0,Y 193.438,Z 425.008,A -85,B 0,C 180,E1 -21780.001,E2 -21780.001} C_VEL
LIN {X 0,Y 192.974,Z 425.073,A -85,B 0,C 180,E1 -21784.178,E2 -21784.178} C_VEL
LIN {X 0,Y 193.054,Z 425.024,A -85,B 0,C 180,E1 -21788.374,E2 -21788.374} C_VEL
LIN {X 0,Y 192.845,Z 425.081,A -85,B 0,C 180,E1 -21792.631,E2 -21792.631} C_VEL
LIN {X 0,Y 192.75,Z 425.092,A -85,B 0,C 180,E1 -21796.96,E2 -21796.96} C_VEL
LIN {X 0,Y 192.629,Z 425.11,A -85,B 0,C 180,E1 -21801.399,E2 -21801.399} C_VEL
LIN {X 0,Y 192.657,Z 425.11,A -85,B 0,C 180,E1 -21804.226,E2 -21804.226} C_VEL
LIN {X 0,Y 192.637,Z 425.08,A -85,B 0,C 180,E1 -21808.891,E2 -21808.891} C_VEL
LIN {X 0,Y 192.591,Z 425.115,A -85,B 0,C 180,E1 -21813.188,E2 -21813.188} C_VEL
LIN {X 0,Y 192.545,Z 425.098,A -85,B 0,C 180,E1 -21818.354,E2 -21818.354} C_VEL
LIN {X 0,Y 192.512,Z 425.125,A -85,B 0,C 180,E1 -21823.106,E2 -21823.106} C_VEL
LIN {X 0,Y 192.544,Z 425.115,A -85,B 0,C 180,E1 -21826.889,E2 -21826.889} C_VEL
LIN {X 0,Y 192.572,Z 425.111,A -85,B 0,C 180,E1 -21831.656,E2 -21831.656} C_VEL
LIN {X 0,Y 192.589,Z 425.187,A -85,B 0,C 180,E1 -21835.48,E2 -21835.48} C_VEL
LIN {X 0,Y 193.627,Z 428.03,A -85,B 0,C 180,E1 -21835.843,E2 -21835.843} C_VEL
LIN {X 0,Y 195.117,Z 430.018,A -85,B 0,C 180,E1 -21836.267,E2 -21836.267} C_VEL
LIN {X 0,Y 200.935,Z 440.637,A -85,B 0,C 180,E1 -21838.216,E2 -21838.216} C_VEL
LIN {X 0,Y 205.511,Z 450.735,A -85,B 0,C 180,E1 -21840.127,E2 -21840.127} C_VEL
LIN {X 0,Y 208.669,Z 459.674,A -85,B 0,C 180,E1 -21841.87,E2 -21841.87} C_VEL
LIN {X 0,Y 210.709,Z 466.748,A -85,B 0,C 180,E1 -21843.339,E2 -21843.339} C_VEL
LIN {X 0,Y 208.776,Z 477.826,A -85,B 0,C 180,E1 -21845.118,E2 -21845.118} C_VEL
LIN {X 0,Y 206.545,Z 487.341,A -85,B 0,C 180,E1 -21847.012,E2 -21847.012} C_VEL
LIN {X 0,Y 204.069,Z 496.68,A -85,B 0,C 180,E1 -21849.331,E2 -21849.331} C_VEL
LIN {X 0,Y 201.715,Z 504.488,A -85,B 0,C 180,E1 -21851.728,E2 -21851.728} C_VEL
LIN {X 0,Y 199.423,Z 512.117,A -85,B 0,C 180,E1 -21854.676,E2 -21854.676} C_VEL
LIN {X 0,Y 197.441,Z 518.21,A -85,B 0,C 180,E1 -21857.671,E2 -21857.671} C_VEL
LIN {X 0,Y 195.94,Z 523.026,A -85,B 0,C 180,E1 -21860.714,E2 -21860.714} C_VEL
LIN {X 0,Y 194.586,Z 526.774,A -85,B 0,C 180,E1 -21863.782,E2 -21863.782} C_VEL
LIN {X 0,Y 193.571,Z 530.208,A -85,B 0,C 180,E1 -21867.922,E2 -21867.922} C_VEL
LIN {X 0,Y 193.401,Z 531.296,A -85,B 0,C 180,E1 -21870.002,E2 -21870.002} C_VEL
LIN {X 0,Y 193.407,Z 531.972,A -85,B 0,C 180,E1 -21872.085,E2 -21872.085} C_VEL
LIN {X 0,Y 193.416,Z 532.284,A -85,B 0,C 180,E1 -21876.26,E2 -21876.26} C_VEL
LIN {X 0,Y 193.945,Z 531.796,A -85,B 0,C 180,E1 -21878.336,E2 -21878.336} C_VEL
LIN {X 0,Y 195.696,Z 529.627,A -85,B 0,C 180,E1 -21882.446,E2 -21882.446} C_VEL
LIN {X 0,Y 197.305,Z 526.58,A -85,B 0,C 180,E1 -21885.898,E2 -21885.898} C_VEL
LIN {X 0,Y 199.626,Z 521.813,A -85,B 0,C 180,E1 -21889.542,E2 -21889.542} C_VEL
LIN {X 0,Y 202.239,Z 515.658,A -85,B 0,C 180,E1 -21893.016,E2 -21893.016} C_VEL
LIN {X 0,Y 205.011,Z 508.832,A -85,B 0,C 180,E1 -21895.92,E2 -21895.92} C_VEL
LIN {X 0,Y 208.158,Z 500.423,A -85,B 0,C 180,E1 -21898.705,E2 -21898.705} C_VEL
LIN {X 0,Y 211.122,Z 491.448,A -85,B 0,C 180,E1 -21901.065,E2 -21901.065} C_VEL
LIN {X 0,Y 213.861,Z 481.644,A -85,B 0,C 180,E1 -21903.118,E2 -21903.118} C_VEL
LIN {X 0,Y 215.432,Z 474.958,A -85,B 0,C 180,E1 -21904.287,E2 -21904.287} C_VEL
LIN {X 0,Y 215.174,Z 472.559,A -85,B 0,C 180,E1 -21904.828,E2 -21904.828} C_VEL
LIN {X 0,Y 212.471,Z 463.342,A -85,B 0,C 180,E1 -21907.06,E2 -21907.06} C_VEL
LIN {X 0,Y 208.818,Z 453.849,A -85,B 0,C 180,E1 -21909.276,E2 -21909.276} C_VEL
LIN {X 0,Y 204.008,Z 444.052,A -85,B 0,C 180,E1 -21911.564,E2 -21911.564} C_VEL
LIN {X 0,Y 199.094,Z 435.829,A -85,B 0,C 180,E1 -21913.551,E2 -21913.551} C_VEL
LIN {X 0,Y 194.269,Z 428.928,A -85,B 0,C 180,E1 -21915.316,E2 -21915.316} C_VEL
LIN {X 0,Y 193.103,Z 427.17,A -85,B 0,C 180,E1 -21915.797,E2 -21915.797} C_VEL
LIN {X 0,Y 192.528,Z 425.128,A -85,B 0,C 180,E1 -21917.233,E2 -21917.233} C_VEL
LIN {X 0,Y 192.557,Z 425.078,A -85,B 0,C 180,E1 -21921.649,E2 -21921.649} C_VEL
LIN {X 0,Y 192.604,Z 425.099,A -85,B 0,C 180,E1 -21926.814,E2 -21926.814} C_VEL
LIN {X 0,Y 192.673,Z 425.095,A -85,B 0,C 180,E1 -21931.175,E2 -21931.175} C_VEL
LIN {X 0,Y 196.495,Z 439.655,A -85,B 0,C 180,E1 -21933.406,E2 -21933.406} C_VEL
LIN {X 0,Y 200.122,Z 453.634,A -85,B 0,C 180,E1 -21935.939,E2 -21935.939} C_VEL
LIN {X 0,Y 200.583,Z 455.443,A -85,B 0,C 180,E1 -21936.292,E2 -21936.292} C_VEL
LIN {X 0,Y 198.738,Z 468.075,A -85,B 0,C 180,E1 -21938.747,E2 -21938.747} C_VEL
LIN {X 0,Y 196.775,Z 480.932,A -85,B 0,C 180,E1 -21941.789,E2 -21941.789} C_VEL
LIN {X 0,Y 195.243,Z 491.803,A -85,B 0,C 180,E1 -21944.872,E2 -21944.872} C_VEL
LIN {X 0,Y 193.902,Z 502.383,A -85,B 0,C 180,E1 -21948.47,E2 -21948.47} C_VEL
LIN {X 0,Y 193.155,Z 510.198,A -85,B 0,C 180,E1 -21951.631,E2 -21951.631} C_VEL
LIN {X 0,Y 192.542,Z 518.843,A -85,B 0,C 180,E1 -21955.813,E2 -21955.813} C_VEL
LIN {X 0,Y 192.814,Z 524.196,A -85,B 0,C 180,E1 -21958.955,E2 -21958.955} C_VEL
LIN {X 0,Y 193.364,Z 530.108,A -85,B 0,C 180,E1 -21963.125,E2 -21963.125} C_VEL
LIN {X 0,Y 194.328,Z 533.663,A -85,B 0,C 180,E1 -21966.228,E2 -21966.228} C_VEL
LIN {X 0,Y 196.392,Z 537.339,A -85,B 0,C 180,E1 -21970.307,E2 -21970.307} C_VEL
LIN {X 0,Y 199.4,Z 539.847,A -85,B 0,C 180,E1 -21974.283,E2 -21974.283} C_VEL
LIN {X 0,Y 203.288,Z 541.225,A -85,B 0,C 180,E1 -21978.128,E2 -21978.128} C_VEL
LIN {X 0,Y 207.914,Z 541.55,A -85,B 0,C 180,E1 -21981.828,E2 -21981.828} C_VEL
LIN {X 0,Y 213.499,Z 540.803,A -85,B 0,C 180,E1 -21985.336,E2 -21985.336} C_VEL
LIN {X 0,Y 219.933,Z 538.999,A -85,B 0,C 180,E1 -21988.641,E2 -21988.641} C_VEL
LIN {X 0,Y 227.214,Z 536.1,A -85,B 0,C 180,E1 -21991.724,E2 -21991.724} C_VEL
LIN {X 0,Y 235.164,Z 532.15,A -85,B 0,C 180,E1 -21994.598,E2 -21994.598} C_VEL
LIN {X 0,Y 243.789,Z 527.06,A -85,B 0,C 180,E1 -21997.257,E2 -21997.257} C_VEL
LIN {X 0,Y 246.05,Z 525.593,A -85,B 0,C 180,E1 -21997.887,E2 -21997.887} C_VEL
LIN {X 0,Y 247.908,Z 524.416,A -85,B 0,C 180,E1 -21998.585,E2 -21998.585} C_VEL
LIN {X 0,Y 247.601,Z 525.149,A -85,B 0,C 180,E1 -21999.968,E2 -21999.968} C_VEL
LIN {X 0,Y 246.68,Z 526.337,A -85,B 0,C 180,E1 -22000.94,E2 -22000.94} C_VEL
LIN {X 0,Y 241.866,Z 531.638,A -85,B 0,C 180,E1 -22003.41,E2 -22003.41} C_VEL
LIN {X 0,Y 236.075,Z 538.144,A -85,B 0,C 180,E1 -22006.077,E2 -22006.077} C_VEL
LIN {X 0,Y 229.422,Z 545.243,A -85,B 0,C 180,E1 -22008.803,E2 -22008.803} C_VEL
LIN {X 0,Y 219.605,Z 554.653,A -85,B 0,C 180,E1 -22012.549,E2 -22012.549} C_VEL
LIN {X 0,Y 214.191,Z 559.716,A -85,B 0,C 180,E1 -22014.954,E2 -22014.954} C_VEL
LIN {X 0,Y 208.224,Z 564.886,A -85,B 0,C 180,E1 -22017.831,E2 -22017.831} C_VEL
LIN {X 0,Y 201.767,Z 570.673,A -85,B 0,C 180,E1 -22021.948,E2 -22021.948} C_VEL
LIN {X 0,Y 197.551,Z 574.483,A -85,B 0,C 180,E1 -22025.533,E2 -22025.533} C_VEL
LIN {X 0,Y 195.494,Z 575.896,A -85,B 0,C 180,E1 -22027.101,E2 -22027.101} C_VEL
LIN {X 0,Y 190.766,Z 577.571,A -85,B 0,C 180,E1 -22029.642,E2 -22029.642} C_VEL
LIN {X 0,Y 186.531,Z 578.598,A -85,B 0,C 180,E1 -22032.338,E2 -22032.338} C_VEL
LIN {X 0,Y 185.283,Z 579.096,A -85,B 0,C 180,E1 -22034.102,E2 -22034.102} C_VEL
LIN {X 0,Y 184.751,Z 580.04,A -85,B 0,C 180,E1 -22036.804,E2 -22036.804} C_VEL
LIN {X 0,Y 184.479,Z 583.877,A -85,B 0,C 180,E1 -22041.233,E2 -22041.233} C_VEL
LIN {X 0,Y 184.715,Z 585.132,A -85,B 0,C 180,E1 -22043.443,E2 -22043.443} C_VEL
LIN {X 0,Y 185.131,Z 585.976,A -85,B 0,C 180,E1 -22045.643,E2 -22045.643} C_VEL
LIN {X 0,Y 185.566,Z 586.401,A -85,B 0,C 180,E1 -22047.827,E2 -22047.827} C_VEL
LIN {X 0,Y 186.185,Z 586.423,A -85,B 0,C 180,E1 -22049.998,E2 -22049.998} C_VEL
LIN {X 0,Y 185.671,Z 585.804,A -85,B 0,C 180,E1 -22052.167,E2 -22052.167} C_VEL
LIN {X 0,Y 185.288,Z 584.771,A -85,B 0,C 180,E1 -22054.348,E2 -22054.348} C_VEL
LIN {X 0,Y 184.934,Z 583.307,A -85,B 0,C 180,E1 -22056.544,E2 -22056.544} C_VEL
LIN {X 0,Y 184.633,Z 580.227,A -85,B 0,C 180,E1 -22059.86,E2 -22059.86} C_VEL
LIN {X 0,Y 184.731,Z 576.068,A -85,B 0,C 180,E1 -22063.192,E2 -22063.192} C_VEL
LIN {X 0,Y 185.66,Z 569.713,A -85,B 0,C 180,E1 -22067.057,E2 -22067.057} C_VEL
LIN {X 0,Y 187.003,Z 563.508,A -85,B 0,C 180,E1 -22070.024,E2 -22070.024} C_VEL
LIN {X 0,Y 188.921,Z 555.817,A -85,B 0,C 180,E1 -22072.99,E2 -22072.99} C_VEL
LIN {X 0,Y 191.063,Z 547.41,A -85,B 0,C 180,E1 -22075.605,E2 -22075.605} C_VEL
LIN {X 0,Y 192.773,Z 540.426,A -85,B 0,C 180,E1 -22077.402,E2 -22077.402} C_VEL
LIN {X 0,Y 193.395,Z 528.636,A -85,B 0,C 180,E1 -22080.124,E2 -22080.124} C_VEL
LIN {X 0,Y 193.837,Z 516.779,A -85,B 0,C 180,E1 -22082.327,E2 -22082.327} C_VEL
LIN {X 0,Y 194.118,Z 503.861,A -85,B 0,C 180,E1 -22084.227,E2 -22084.227} C_VEL
LIN {X 0,Y 194.174,Z 490.565,A -85,B 0,C 180,E1 -22085.704,E2 -22085.704} C_VEL
LIN {X 0,Y 193.774,Z 479.316,A -85,B 0,C 180,E1 -22086.643,E2 -22086.643} C_VEL
LIN {X 0,Y 190.753,Z 463.82,A -85,B 0,C 180,E1 -22088.047,E2 -22088.047} C_VEL
LIN {X 0,Y 190.161,Z 451.074,A -85,B 0,C 180,E1 -22090.636,E2 -22090.636} C_VEL
LIN {X 0,Y 189.69,Z 445.948,A -85,B 0,C 180,E1 -22091.824,E2 -22091.824} C_VEL
LIN {X 0,Y 189.407,Z 443.4,A -85,B 0,C 180,E1 -22093.654,E2 -22093.654} C_VEL
LIN {X 0,Y 187.618,Z 435.708,A -85,B 0,C 180,E1 -22099.398,E2 -22099.398} C_VEL
LIN {X 0,Y 186.334,Z 429.53,A -85,B 0,C 180,E1 -22104.225,E2 -22104.225} C_VEL
LIN {X 0,Y 185.656,Z 425.98,A -85,B 0,C 180,E1 -22107.134,E2 -22107.134} C_VEL
LIN {X 0,Y 185.574,Z 425.987,A -85,B 0,C 180,E1 -22110.574,E2 -22110.574} C_VEL
LIN {X 0,Y 185.579,Z 425.986,A -85,B 0,C 180,E1 -22115.382,E2 -22115.382} C_VEL
LIN {X 0,Y 185.666,Z 425.978,A -85,B 0,C 180,E1 -22121.133,E2 -22121.133} C_VEL
LIN {X 0,Y 185.756,Z 425.971,A -85,B 0,C 180,E1 -22126.88,E2 -22126.88} C_VEL
LIN {X 0,Y 186,Z 425.936,A -85,B 0,C 180,E1 -22131.308,E2 -22131.308} C_VEL
LIN {X 0,Y 186.201,Z 425.916,A -85,B 0,C 180,E1 -22137.837,E2 -22137.837} C_VEL
LIN {X 0,Y 186.401,Z 425.884,A -85,B 0,C 180,E1 -22140.001,E2 -22140.001} C_VEL
LIN {X 0,Y 185.921,Z 425.951,A -85,B 0,C 180,E1 -22144.336,E2 -22144.336} C_VEL
LIN {X 0,Y 186.001,Z 425.9,A -85,B 0,C 180,E1 -22148.694,E2 -22148.694} C_VEL
LIN {X 0,Y 185.757,Z 425.968,A -85,B 0,C 180,E1 -22153.122,E2 -22153.122} C_VEL
LIN {X 0,Y 185.683,Z 425.973,A -85,B 0,C 180,E1 -22157.626,E2 -22157.626} C_VEL
LIN {X 0,Y 185.589,Z 425.983,A -85,B 0,C 180,E1 -22162.253,E2 -22162.253} C_VEL
LIN {X 0,Y 185.554,Z 425.983,A -85,B 0,C 180,E1 -22167.034,E2 -22167.034} C_VEL
LIN {X 0,Y 185.571,Z 425.956,A -85,B 0,C 180,E1 -22169.495,E2 -22169.495} C_VEL
LIN {X 0,Y 185.493,Z 426.002,A -85,B 0,C 180,E1 -22174.634,E2 -22174.634} C_VEL
LIN {X 0,Y 185.499,Z 425.977,A -85,B 0,C 180,E1 -22177.316,E2 -22177.316} C_VEL
LIN {X 0,Y 185.466,Z 425.999,A -85,B 0,C 180,E1 -22180.727,E2 -22180.727} C_VEL
LIN {X 0,Y 185.505,Z 425.984,A -85,B 0,C 180,E1 -22186.042,E2 -22186.042} C_VEL
LIN {X 0,Y 185.5,Z 425.992,A -85,B 0,C 180,E1 -22189.907,E2 -22189.907} C_VEL
LIN {X 0,Y 185.598,Z 426.195,A -85,B 0,C 180,E1 -22193.856,E2 -22193.856} C_VEL
LIN {X 0,Y 186.701,Z 429.076,A -85,B 0,C 180,E1 -22194.294,E2 -22194.294} C_VEL
LIN {X 0,Y 188.237,Z 431.232,A -85,B 0,C 180,E1 -22194.774,E2 -22194.774} C_VEL
LIN {X 0,Y 194.235,Z 441.818,A -85,B 0,C 180,E1 -22196.91,E2 -22196.91} C_VEL
LIN {X 0,Y 198.482,Z 451.053,A -85,B 0,C 180,E1 -22198.77,E2 -22198.77} C_VEL
LIN {X 0,Y 201.749,Z 459.643,A -85,B 0,C 180,E1 -22200.563,E2 -22200.563} C_VEL
LIN {X 0,Y 204.276,Z 468.452,A -85,B 0,C 180,E1 -22202.479,E2 -22202.479} C_VEL
LIN {X 0,Y 203.909,Z 471.878,A -85,B 0,C 180,E1 -22203.053,E2 -22203.053} C_VEL
LIN {X 0,Y 201.832,Z 481.826,A -85,B 0,C 180,E1 -22204.809,E2 -22204.809} C_VEL
LIN {X 0,Y 199.397,Z 491.432,A -85,B 0,C 180,E1 -22206.905,E2 -22206.905} C_VEL
LIN {X 0,Y 196.478,Z 501.17,A -85,B 0,C 180,E1 -22209.591,E2 -22209.591} C_VEL
LIN {X 0,Y 193.843,Z 509.656,A -85,B 0,C 180,E1 -22212.598,E2 -22212.598} C_VEL
LIN {X 0,Y 191.828,Z 515.424,A -85,B 0,C 180,E1 -22215.142,E2 -22215.142} C_VEL
LIN {X 0,Y 190.081,Z 521.045,A -85,B 0,C 180,E1 -22218.269,E2 -22218.269} C_VEL
LIN {X 0,Y 188.478,Z 525.491,A -85,B 0,C 180,E1 -22221.425,E2 -22221.425} C_VEL
LIN {X 0,Y 187.604,Z 527.837,A -85,B 0,C 180,E1 -22223.55,E2 -22223.55} C_VEL
LIN {X 0,Y 186.551,Z 531.252,A -85,B 0,C 180,E1 -22227.843,E2 -22227.843} C_VEL
LIN {X 0,Y 186.373,Z 532.322,A -85,B 0,C 180,E1 -22230.002,E2 -22230.002} C_VEL
LIN {X 0,Y 186.383,Z 532.99,A -85,B 0,C 180,E1 -22232.163,E2 -22232.163} C_VEL
LIN {X 0,Y 186.424,Z 533.283,A -85,B 0,C 180,E1 -22236.496,E2 -22236.496} C_VEL
LIN {X 0,Y 186.988,Z 532.779,A -85,B 0,C 180,E1 -22238.649,E2 -22238.649} C_VEL
LIN {X 0,Y 188.836,Z 530.591,A -85,B 0,C 180,E1 -22242.905,E2 -22242.905} C_VEL
LIN {X 0,Y 190.519,Z 527.561,A -85,B 0,C 180,E1 -22246.439,E2 -22246.439} C_VEL
LIN {X 0,Y 192.977,Z 522.731,A -85,B 0,C 180,E1 -22250.244,E2 -22250.244} C_VEL
LIN {X 0,Y 195.769,Z 516.547,A -85,B 0,C 180,E1 -22253.822,E2 -22253.822} C_VEL
LIN {X 0,Y 198.699,Z 509.683,A -85,B 0,C 180,E1 -22256.808,E2 -22256.808} C_VEL
LIN {X 0,Y 202,Z 501.243,A -85,B 0,C 180,E1 -22259.666,E2 -22259.666} C_VEL
LIN {X 0,Y 205.122,Z 492.223,A -85,B 0,C 180,E1 -22262.08,E2 -22262.08} C_VEL
LIN {X 0,Y 207.979,Z 482.353,A -85,B 0,C 180,E1 -22264.182,E2 -22264.182} C_VEL
LIN {X 0,Y 209.232,Z 477.109,A -85,B 0,C 180,E1 -22265.137,E2 -22265.137} C_VEL
LIN {X 0,Y 208.978,Z 474.495,A -85,B 0,C 180,E1 -22265.768,E2 -22265.768} C_VEL
LIN {X 0,Y 206.058,Z 464.511,A -85,B 0,C 180,E1 -22268.328,E2 -22268.328} C_VEL
LIN {X 0,Y 202.456,Z 455.341,A -85,B 0,C 180,E1 -22270.629,E2 -22270.629} C_VEL
LIN {X 0,Y 198.106,Z 446.404,A -85,B 0,C 180,E1 -22272.877,E2 -22272.877} C_VEL
LIN {X 0,Y 193.116,Z 438.152,A -85,B 0,C 180,E1 -22275.069,E2 -22275.069} C_VEL
LIN {X 0,Y 186.251,Z 428.392,A -85,B 0,C 180,E1 -22277.837,E2 -22277.837} C_VEL
LIN {X 0,Y 185.482,Z 425.967,A -85,B 0,C 180,E1 -22279.679,E2 -22279.679} C_VEL
LIN {X 0,Y 185.512,Z 425.961,A -85,B 0,C 180,E1 -22282.712,E2 -22282.712} C_VEL
LIN {X 0,Y 185.55,Z 425.951,A -85,B 0,C 180,E1 -22287.975,E2 -22287.975} C_VEL
LIN {X 0,Y 185.59,Z 425.926,A -85,B 0,C 180,E1 -22290.759,E2 -22290.759} C_VEL
LIN {X 0,Y 189.735,Z 441.863,A -85,B 0,C 180,E1 -22293.348,E2 -22293.348} C_VEL
LIN {X 0,Y 193.255,Z 455.435,A -85,B 0,C 180,E1 -22295.916,E2 -22295.916} C_VEL
LIN {X 0,Y 193.535,Z 456.821,A -85,B 0,C 180,E1 -22296.192,E2 -22296.192} C_VEL
LIN {X 0,Y 191.326,Z 470.598,A -85,B 0,C 180,E1 -22299.013,E2 -22299.013} C_VEL
LIN {X 0,Y 189.408,Z 483.196,A -85,B 0,C 180,E1 -22302.174,E2 -22302.174} C_VEL
LIN {X 0,Y 187.915,Z 493.868,A -85,B 0,C 180,E1 -22305.377,E2 -22305.377} C_VEL
LIN {X 0,Y 186.648,Z 504.381,A -85,B 0,C 180,E1 -22309.148,E2 -22309.148} C_VEL
LIN {X 0,Y 185.844,Z 511.974,A -85,B 0,C 180,E1 -22312.394,E2 -22312.394} C_VEL
LIN {X 0,Y 185.478,Z 520.503,A -85,B 0,C 180,E1 -22316.741,E2 -22316.741} C_VEL
LIN {X 0,Y 185.764,Z 525.811,A -85,B 0,C 180,E1 -22319.999,E2 -22319.999} C_VEL
LIN {X 0,Y 186.554,Z 531.673,A -85,B 0,C 180,E1 -22324.321,E2 -22324.321} C_VEL
LIN {X 0,Y 188.215,Z 536.247,A -85,B 0,C 180,E1 -22328.589,E2 -22328.589} C_VEL
LIN {X 0,Y 190.905,Z 539.622,A -85,B 0,C 180,E1 -22332.761,E2 -22332.761} C_VEL
LIN {X 0,Y 194.504,Z 541.863,A -85,B 0,C 180,E1 -22336.801,E2 -22336.801} C_VEL
LIN {X 0,Y 199.024,Z 543,A -85,B 0,C 180,E1 -22340.678,E2 -22340.678} C_VEL
LIN {X 0,Y 204.375,Z 543.099,A -85,B 0,C 180,E1 -22344.371,E2 -22344.371} C_VEL
LIN {X 0,Y 210.623,Z 542.166,A -85,B 0,C 180,E1 -22347.849,E2 -22347.849} C_VEL
LIN {X 0,Y 217.75,Z 540.195,A -85,B 0,C 180,E1 -22351.091,E2 -22351.091} C_VEL
LIN {X 0,Y 225.67,Z 537.168,A -85,B 0,C 180,E1 -22354.095,E2 -22354.095} C_VEL
LIN {X 0,Y 234.281,Z 533.086,A -85,B 0,C 180,E1 -22356.867,E2 -22356.867} C_VEL
LIN {X 0,Y 241.148,Z 529.35,A -85,B 0,C 180,E1 -22358.799,E2 -22358.799} C_VEL
LIN {X 0,Y 241.746,Z 529.313,A -85,B 0,C 180,E1 -22359.76,E2 -22359.76} C_VEL
LIN {X 0,Y 240.6,Z 530.533,A -85,B 0,C 180,E1 -22360.581,E2 -22360.581} C_VEL
LIN {X 0,Y 235.294,Z 535.777,A -85,B 0,C 180,E1 -22363.087,E2 -22363.087} C_VEL
LIN {X 0,Y 230.038,Z 541.038,A -85,B 0,C 180,E1 -22365.355,E2 -22365.355} C_VEL
LIN {X 0,Y 224.229,Z 546.57,A -85,B 0,C 180,E1 -22367.631,E2 -22367.631} C_VEL
LIN {X 0,Y 214.042,Z 555.363,A -85,B 0,C 180,E1 -22371.399,E2 -22371.399} C_VEL
LIN {X 0,Y 208.427,Z 560.066,A -85,B 0,C 180,E1 -22373.835,E2 -22373.835} C_VEL
LIN {X 0,Y 201.355,Z 565.617,A -85,B 0,C 180,E1 -22377.246,E2 -22377.246} C_VEL
LIN {X 0,Y 194.208,Z 571.299,A -85,B 0,C 180,E1 -22381.935,E2 -22381.935} C_VEL
LIN {X 0,Y 189.827,Z 574.886,A -85,B 0,C 180,E1 -22385.965,E2 -22385.965} C_VEL
LIN {X 0,Y 186.805,Z 577.522,A -85,B 0,C 180,E1 -22390.206,E2 -22390.206} C_VEL
LIN {X 0,Y 185.283,Z 579.096,A -85,B 0,C 180,E1 -22394.102,E2 -22394.102} C_VEL
LIN {X 0,Y 184.217,Z 579.888,A -85,B 0,C 180,E1 -22395.884,E2 -22395.884} C_VEL
LIN {X 0,Y 180.996,Z 581.653,A -85,B 0,C 180,E1 -22398.773,E2 -22398.773} C_VEL
LIN {X 0,Y 178.558,Z 583.172,A -85,B 0,C 180,E1 -22401.144,E2 -22401.144} C_VEL
LIN {X 0,Y 177.677,Z 584.067,A -85,B 0,C 180,E1 -22403.006,E2 -22403.006} C_VEL
LIN {X 0,Y 177.682,Z 584.299,A -85,B 0,C 180,E1 -22403.638,E2 -22403.638} C_VEL
LIN {X 0,Y 178.05,Z 584.973,A -85,B 0,C 180,E1 -22405.47,E2 -22405.47} C_VEL
LIN {X 0,Y 178.487,Z 585.393,A -85,B 0,C 180,E1 -22407.741,E2 -22407.741} C_VEL
LIN {X 0,Y 179.135,Z 585.407,A -85,B 0,C 180,E1 -22409.998,E2 -22409.998} C_VEL
LIN {X 0,Y 178.592,Z 584.772,A -85,B 0,C 180,E1 -22412.253,E2 -22412.253} C_VEL
LIN {X 0,Y 178.208,Z 583.729,A -85,B 0,C 180,E1 -22414.521,E2 -22414.521} C_VEL
LIN {X 0,Y 177.653,Z 580.848,A -85,B 0,C 180,E1 -22418.507,E2 -22418.507} C_VEL
LIN {X 0,Y 177.588,Z 576.477,A -85,B 0,C 180,E1 -22422.569,E2 -22422.569} C_VEL
LIN {X 0,Y 178.232,Z 571.529,A -85,B 0,C 180,E1 -22426.02,E2 -22426.02} C_VEL
LIN {X 0,Y 179.486,Z 565.361,A -85,B 0,C 180,E1 -22429.407,E2 -22429.407} C_VEL
LIN {X 0,Y 181.482,Z 557.61,A -85,B 0,C 180,E1 -22432.781,E2 -22432.781} C_VEL
LIN {X 0,Y 183.648,Z 549.798,A -85,B 0,C 180,E1 -22435.498,E2 -22435.498} C_VEL
LIN {X 0,Y 185.908,Z 541.34,A -85,B 0,C 180,E1 -22437.89,E2 -22437.89} C_VEL
LIN {X 0,Y 186.693,Z 530.228,A -85,B 0,C 180,E1 -22440.641,E2 -22440.641} C_VEL
LIN {X 0,Y 187.293,Z 518.8,A -85,B 0,C 180,E1 -22442.96,E2 -22442.96} C_VEL
LIN {X 0,Y 187.814,Z 506.989,A -85,B 0,C 180,E1 -22444.882,E2 -22444.882} C_VEL
LIN {X 0,Y 188.082,Z 493.68,A -85,B 0,C 180,E1 -22446.546,E2 -22446.546} C_VEL
LIN {X 0,Y 187.96,Z 481.663,A -85,B 0,C 180,E1 -22447.67,E2 -22447.67} C_VEL
LIN {X 0,Y 185.265,Z 466.586,A -85,B 0,C 180,E1 -22449.117,E2 -22449.117} C_VEL
LIN {X 0,Y 184.452,Z 462.531,A -85,B 0,C 180,E1 -22449.554,E2 -22449.554} C_VEL
LIN {X 0,Y 183.913,Z 452.209,A -85,B 0,C 180,E1 -22451.827,E2 -22451.827} C_VEL
LIN {X 0,Y 183.663,Z 448.987,A -85,B 0,C 180,E1 -22452.557,E2 -22452.557} C_VEL
LIN {X 0,Y 182.03,Z 442.688,A -85,B 0,C 180,E1 -22454.41,E2 -22454.41} C_VEL
LIN {X 0,Y 180.752,Z 437.244,A -85,B 0,C 180,E1 -22458.625,E2 -22458.625} C_VEL
LIN {X 0,Y 179.342,Z 430.576,A -85,B 0,C 180,E1 -22463.998,E2 -22463.998} C_VEL
LIN {X 0,Y 178.631,Z 426.855,A -85,B 0,C 180,E1 -22467.251,E2 -22467.251} C_VEL
LIN {X 0,Y 178.48,Z 426.874,A -85,B 0,C 180,E1 -22471.802,E2 -22471.802} C_VEL
LIN {X 0,Y 178.503,Z 426.874,A -85,B 0,C 180,E1 -22476.814,E2 -22476.814} C_VEL
LIN {X 0,Y 178.642,Z 426.858,A -85,B 0,C 180,E1 -22481.656,E2 -22481.656} C_VEL
LIN {X 0,Y 178.674,Z 426.851,A -85,B 0,C 180,E1 -22486.35,E2 -22486.35} C_VEL
LIN {X 0,Y 178.929,Z 426.814,A -85,B 0,C 180,E1 -22490.961,E2 -22490.961} C_VEL
LIN {X 0,Y 179.147,Z 426.795,A -85,B 0,C 180,E1 -22497.752,E2 -22497.752} C_VEL
LIN {X 0,Y 179.364,Z 426.76,A -85,B 0,C 180,E1 -22500.001,E2 -22500.001} C_VEL
LIN {X 0,Y 178.869,Z 426.828,A -85,B 0,C 180,E1 -22504.508,E2 -22504.508} C_VEL
LIN {X 0,Y 178.93,Z 426.779,A -85,B 0,C 180,E1 -22509.04,E2 -22509.04} C_VEL
LIN {X 0,Y 178.679,Z 426.853,A -85,B 0,C 180,E1 -22513.651,E2 -22513.651} C_VEL
LIN {X 0,Y 178.642,Z 426.853,A -85,B 0,C 180,E1 -22518.345,E2 -22518.345} C_VEL
LIN {X 0,Y 178.504,Z 426.868,A -85,B 0,C 180,E1 -22523.187,E2 -22523.187} C_VEL
LIN {X 0,Y 178.478,Z 426.846,A -85,B 0,C 180,E1 -22528.199,E2 -22528.199} C_VEL
LIN {X 0,Y 178.471,Z 426.843,A -85,B 0,C 180,E1 -22530.793,E2 -22530.793} C_VEL
LIN {X 0,Y 178.478,Z 426.877,A -85,B 0,C 180,E1 -22534.221,E2 -22534.221} C_VEL
LIN {X 0,Y 178.39,Z 426.861,A -85,B 0,C 180,E1 -22539.077,E2 -22539.077} C_VEL
LIN {X 0,Y 178.404,Z 426.887,A -85,B 0,C 180,E1 -22542.044,E2 -22542.044} C_VEL
LIN {X 0,Y 178.421,Z 426.863,A -85,B 0,C 180,E1 -22545.156,E2 -22545.156} C_VEL
LIN {X 0,Y 178.428,Z 426.885,A -85,B 0,C 180,E1 -22548.451,E2 -22548.451} C_VEL
LIN {X 0,Y 178.476,Z 426.961,A -85,B 0,C 180,E1 -22551.862,E2 -22551.862} C_VEL
LIN {X 0,Y 178.571,Z 427.532,A -85,B 0,C 180,E1 -22552.127,E2 -22552.127} C_VEL
LIN {X 0,Y 179.741,Z 430.107,A -85,B 0,C 180,E1 -22552.576,E2 -22552.576} C_VEL
LIN {X 0,Y 181.276,Z 432.058,A -85,B 0,C 180,E1 -22553.087,E2 -22553.087} C_VEL
LIN {X 0,Y 187.609,Z 442.987,A -85,B 0,C 180,E1 -22555.503,E2 -22555.503} C_VEL
LIN {X 0,Y 191.795,Z 451.914,A -85,B 0,C 180,E1 -22557.438,E2 -22557.438} C_VEL
LIN {X 0,Y 195.521,Z 461.688,A -85,B 0,C 180,E1 -22559.62,E2 -22559.62} C_VEL
LIN {X 0,Y 197.903,Z 470.171,A -85,B 0,C 180,E1 -22561.571,E2 -22561.571} C_VEL
LIN {X 0,Y 198.029,Z 471.594,A -85,B 0,C 180,E1 -22561.878,E2 -22561.878} C_VEL
LIN {X 0,Y 195.526,Z 483.1,A -85,B 0,C 180,E1 -22563.937,E2 -22563.937} C_VEL
LIN {X 0,Y 192.975,Z 492.654,A -85,B 0,C 180,E1 -22566.089,E2 -22566.089} C_VEL
LIN {X 0,Y 189.927,Z 502.346,A -85,B 0,C 180,E1 -22568.854,E2 -22568.854} C_VEL
LIN {X 0,Y 187.165,Z 510.805,A -85,B 0,C 180,E1 -22571.956,E2 -22571.956} C_VEL
LIN {X 0,Y 185.061,Z 516.547,A -85,B 0,C 180,E1 -22574.586,E2 -22574.586} C_VEL
LIN {X 0,Y 183.221,Z 522.144,A -85,B 0,C 180,E1 -22577.823,E2 -22577.823} C_VEL
LIN {X 0,Y 181.538,Z 526.569,A -85,B 0,C 180,E1 -22581.094,E2 -22581.094} C_VEL
LIN {X 0,Y 180.626,Z 528.899,A -85,B 0,C 180,E1 -22583.299,E2 -22583.299} C_VEL
LIN {X 0,Y 179.531,Z 532.296,A -85,B 0,C 180,E1 -22587.759,E2 -22587.759} C_VEL
LIN {X 0,Y 179.359,Z 534.007,A -85,B 0,C 180,E1 -22592.248,E2 -22592.248} C_VEL
LIN {X 0,Y 179.337,Z 534.328,A -85,B 0,C 180,E1 -22594.498,E2 -22594.498} C_VEL
LIN {X 0,Y 179.436,Z 534.28,A -85,B 0,C 180,E1 -22596.75,E2 -22596.75} C_VEL
LIN {X 0,Y 180.945,Z 532.845,A -85,B 0,C 180,E1 -22601.2,E2 -22601.2} C_VEL
LIN {X 0,Y 181.989,Z 531.554,A -85,B 0,C 180,E1 -22603.4,E2 -22603.4} C_VEL
LIN {X 0,Y 183.776,Z 528.516,A -85,B 0,C 180,E1 -22607.046,E2 -22607.046} C_VEL
LIN {X 0,Y 186.372,Z 523.647,A -85,B 0,C 180,E1 -22610.994,E2 -22610.994} C_VEL
LIN {X 0,Y 188.893,Z 518.407,A -85,B 0,C 180,E1 -22614.161,E2 -22614.161} C_VEL
LIN {X 0,Y 191.879,Z 511.81,A -85,B 0,C 180,E1 -22617.25,E2 -22617.25} C_VEL
LIN {X 0,Y 195.316,Z 503.482,A -85,B 0,C 180,E1 -22620.251,E2 -22620.251} C_VEL
LIN {X 0,Y 198.531,Z 494.895,A -85,B 0,C 180,E1 -22622.676,E2 -22622.676} C_VEL
LIN {X 0,Y 201.86,Z 484.302,A -85,B 0,C 180,E1 -22625.065,E2 -22625.065} C_VEL
LIN {X 0,Y 203.136,Z 479.253,A -85,B 0,C 180,E1 -22626.029,E2 -22626.029} C_VEL
LIN {X 0,Y 202.557,Z 475.366,A -85,B 0,C 180,E1 -22627.057,E2 -22627.057} C_VEL
LIN {X 0,Y 199.716,Z 465.814,A -85,B 0,C 180,E1 -22629.665,E2 -22629.665} C_VEL
LIN {X 0,Y 196.296,Z 457.032,A -85,B 0,C 180,E1 -22632.019,E2 -22632.019} C_VEL
LIN {X 0,Y 191.47,Z 447.39,A -85,B 0,C 180,E1 -22634.668,E2 -22634.668} C_VEL
LIN {X 0,Y 186.638,Z 439.627,A -85,B 0,C 180,E1 -22636.959,E2 -22636.959} C_VEL
LIN {X 0,Y 181.897,Z 433.139,A -85,B 0,C 180,E1 -22639.046,E2 -22639.046} C_VEL
LIN {X 0,Y 179.333,Z 429.546,A -85,B 0,C 180,E1 -22640.261,E2 -22640.261} C_VEL
LIN {X 0,Y 178.476,Z 426.835,A -85,B 0,C 180,E1 -22642.523,E2 -22642.523} C_VEL
LIN {X 0,Y 178.492,Z 426.858,A -85,B 0,C 180,E1 -22646.547,E2 -22646.547} C_VEL
LIN {X 0,Y 178.524,Z 426.805,A -85,B 0,C 180,E1 -22650.399,E2 -22650.399} C_VEL
LIN {X 0,Y 182.487,Z 442.118,A -85,B 0,C 180,E1 -22652.952,E2 -22652.952} C_VEL
LIN {X 0,Y 186.048,Z 455.852,A -85,B 0,C 180,E1 -22655.627,E2 -22655.627} C_VEL
LIN {X 0,Y 186.323,Z 458.077,A -85,B 0,C 180,E1 -22656.078,E2 -22656.078} C_VEL
LIN {X 0,Y 184.061,Z 471.827,A -85,B 0,C 180,E1 -22659.024,E2 -22659.024} C_VEL
LIN {X 0,Y 182.305,Z 483.432,A -85,B 0,C 180,E1 -22662.036,E2 -22662.036} C_VEL
LIN {X 0,Y 180.588,Z 495.839,A -85,B 0,C 180,E1 -22665.922,E2 -22665.922} C_VEL
LIN {X 0,Y 179.439,Z 506.187,A -85,B 0,C 180,E1 -22669.848,E2 -22669.848} C_VEL
LIN {X 0,Y 178.443,Z 515.922,A -85,B 0,C 180,E1 -22674.349,E2 -22674.349} C_VEL
LIN {X 0,Y 178.615,Z 523.949,A -85,B 0,C 180,E1 -22678.872,E2 -22678.872} C_VEL
LIN {X 0,Y 179.23,Z 530.453,A -85,B 0,C 180,E1 -22683.371,E2 -22683.371} C_VEL
LIN {X 0,Y 180.724,Z 535.628,A -85,B 0,C 180,E1 -22687.822,E2 -22687.822} C_VEL
LIN {X 0,Y 184.05,Z 540.382,A -85,B 0,C 180,E1 -22693.244,E2 -22693.244} C_VEL
LIN {X 0,Y 187.803,Z 542.94,A -85,B 0,C 180,E1 -22697.42,E2 -22697.42} C_VEL
LIN {X 0,Y 192.535,Z 544.413,A -85,B 0,C 180,E1 -22701.409,E2 -22701.409} C_VEL
LIN {X 0,Y 198.143,Z 544.857,A -85,B 0,C 180,E1 -22705.19,E2 -22705.19} C_VEL
LIN {X 0,Y 204.666,Z 544.285,A -85,B 0,C 180,E1 -22708.734,E2 -22708.734} C_VEL
LIN {X 0,Y 212.067,Z 542.688,A -85,B 0,C 180,E1 -22712.022,E2 -22712.022} C_VEL
LIN {X 0,Y 220.289,Z 540.05,A -85,B 0,C 180,E1 -22715.048,E2 -22715.048} C_VEL
LIN {X 0,Y 229.191,Z 536.398,A -85,B 0,C 180,E1 -22717.827,E2 -22717.827} C_VEL
LIN {X 0,Y 233.873,Z 534.185,A -85,B 0,C 180,E1 -22719.128,E2 -22719.128} C_VEL
LIN {X 0,Y 235.265,Z 533.607,A -85,B 0,C 180,E1 -22719.716,E2 -22719.716} C_VEL
LIN {X 0,Y 229.27,Z 538.925,A -85,B 0,C 180,E1 -22722.406,E2 -22722.406} C_VEL
LIN {X 0,Y 223.157,Z 544.34,A -85,B 0,C 180,E1 -22724.877,E2 -22724.877} C_VEL
LIN {X 0,Y 216.97,Z 549.493,A -85,B 0,C 180,E1 -22727.137,E2 -22727.137} C_VEL
LIN {X 0,Y 208.555,Z 556,A -85,B 0,C 180,E1 -22730.186,E2 -22730.186} C_VEL
LIN {X 0,Y 202.745,Z 560.358,A -85,B 0,C 180,E1 -22732.652,E2 -22732.652} C_VEL
LIN {X 0,Y 195.391,Z 565.524,A -85,B 0,C 180,E1 -22736.113,E2 -22736.113} C_VEL
LIN {X 0,Y 187.929,Z 570.768,A -85,B 0,C 180,E1 -22740.909,E2 -22740.909} C_VEL
LIN {X 0,Y 183.315,Z 573.976,A -85,B 0,C 180,E1 -22745.054,E2 -22745.054} C_VEL
LIN {X 0,Y 180.061,Z 576.394,A -85,B 0,C 180,E1 -22749.511,E2 -22749.511} C_VEL
LIN {X 0,Y 178.063,Z 578.073,A -85,B 0,C 180,E1 -22755.132,E2 -22755.132} C_VEL
LIN {X 0,Y 177.452,Z 581.185,A -85,B 0,C 180,E1 -22758.576,E2 -22758.576} C_VEL
LIN {X 0,Y 177.485,Z 583.454,A -85,B 0,C 180,E1 -22761.864,E2 -22761.864} C_VEL
LIN {X 0,Y 177.682,Z 584.299,A -85,B 0,C 180,E1 -22763.638,E2 -22763.638} C_VEL
LIN {X 0,Y 177.562,Z 584.763,A -85,B 0,C 180,E1 -22764.905,E2 -22764.905} C_VEL
LIN {X 0,Y 176.496,Z 585.039,A -85,B 0,C 180,E1 -22766.798,E2 -22766.798} C_VEL
LIN {X 0,Y 173.637,Z 584.621,A -85,B 0,C 180,E1 -22769.951,E2 -22769.951} C_VEL
LIN {X 0,Y 171.671,Z 583.69,A -85,B 0,C 180,E1 -22772.554,E2 -22772.554} C_VEL
LIN {X 0,Y 171.214,Z 583.049,A -85,B 0,C 180,E1 -22773.889,E2 -22773.889} C_VEL
LIN {X 0,Y 170.715,Z 581.189,A -85,B 0,C 180,E1 -22777.092,E2 -22777.092} C_VEL
LIN {X 0,Y 170.48,Z 578.067,A -85,B 0,C 180,E1 -22780.688,E2 -22780.688} C_VEL
LIN {X 0,Y 170.745,Z 573.87,A -85,B 0,C 180,E1 -22784.295,E2 -22784.295} C_VEL
LIN {X 0,Y 171.94,Z 567.457,A -85,B 0,C 180,E1 -22788.465,E2 -22788.465} C_VEL
LIN {X 0,Y 173.71,Z 560.506,A -85,B 0,C 180,E1 -22791.974,E2 -22791.974} C_VEL
LIN {X 0,Y 176.223,Z 551.931,A -85,B 0,C 180,E1 -22795.384,E2 -22795.384} C_VEL
LIN {X 0,Y 179.035,Z 542.109,A -85,B 0,C 180,E1 -22798.419,E2 -22798.419} C_VEL
LIN {X 0,Y 179.936,Z 532.15,A -85,B 0,C 180,E1 -22801.097,E2 -22801.097} C_VEL
LIN {X 0,Y 180.736,Z 520.962,A -85,B 0,C 180,E1 -22803.588,E2 -22803.588} C_VEL
LIN {X 0,Y 181.507,Z 508.799,A -85,B 0,C 180,E1 -22805.733,E2 -22805.733} C_VEL
LIN {X 0,Y 182.025,Z 496.413,A -85,B 0,C 180,E1 -22807.446,E2 -22807.446} C_VEL
LIN {X 0,Y 182.075,Z 482.896,A -85,B 0,C 180,E1 -22808.866,E2 -22808.866} C_VEL
LIN {X 0,Y 179.914,Z 469.727,A -85,B 0,C 180,E1 -22810.246,E2 -22810.246} C_VEL
LIN {X 0,Y 178.223,Z 461.877,A -85,B 0,C 180,E1 -22811.07,E2 -22811.07} C_VEL
LIN {X 0,Y 177.842,Z 453.588,A -85,B 0,C 180,E1 -22813.015,E2 -22813.015} C_VEL
LIN {X 0,Y 177.235,Z 450.26,A -85,B 0,C 180,E1 -22813.91,E2 -22813.91} C_VEL
LIN {X 0,Y 176.41,Z 446.703,A -85,B 0,C 180,E1 -22814.998,E2 -22814.998} C_VEL
LIN {X 0,Y 174.258,Z 440.679,A -85,B 0,C 180,E1 -22817.111,E2 -22817.111} C_VEL
LIN {X 0,Y 173.916,Z 438.742,A -85,B 0,C 180,E1 -22817.793,E2 -22817.793} C_VEL
LIN {X 0,Y 172.667,Z 433.225,A -85,B 0,C 180,E1 -22822.372,E2 -22822.372} C_VEL
LIN {X 0,Y 171.589,Z 427.732,A -85,B 0,C 180,E1 -22827.133,E2 -22827.133} C_VEL
LIN {X 0,Y 171.411,Z 427.759,A -85,B 0,C 180,E1 -22833.192,E2 -22833.192} C_VEL
LIN {X 0,Y 171.453,Z 427.75,A -85,B 0,C 180,E1 -22838.352,E2 -22838.352} C_VEL
LIN {X 0,Y 171.571,Z 427.732,A -85,B 0,C 180,E1 -22840.871,E2 -22840.871} C_VEL
LIN {X 0,Y 171.586,Z 427.73,A -85,B 0,C 180,E1 -22845.774,E2 -22845.774} C_VEL
LIN {X 0,Y 171.865,Z 427.691,A -85,B 0,C 180,E1 -22850.586,E2 -22850.586} C_VEL
LIN {X 0,Y 171.815,Z 427.698,A -85,B 0,C 180,E1 -22855.308,E2 -22855.308} C_VEL
LIN {X 0,Y 172.327,Z 427.636,A -85,B 0,C 180,E1 -22860.001,E2 -22860.001} C_VEL
LIN {X 0,Y 171.818,Z 427.704,A -85,B 0,C 180,E1 -22864.693,E2 -22864.693} C_VEL
LIN {X 0,Y 171.865,Z 427.658,A -85,B 0,C 180,E1 -22869.415,E2 -22869.415} C_VEL
LIN {X 0,Y 171.602,Z 427.735,A -85,B 0,C 180,E1 -22874.226,E2 -22874.226} C_VEL
LIN {X 0,Y 171.537,Z 427.743,A -85,B 0,C 180,E1 -22879.563,E2 -22879.563} C_VEL
LIN {X 0,Y 171.462,Z 427.751,A -85,B 0,C 180,E1 -22885.618,E2 -22885.618} C_VEL
LIN {X 0,Y 171.433,Z 427.717,A -85,B 0,C 180,E1 -22890.588,E2 -22890.588} C_VEL
LIN {X 0,Y 171.387,Z 427.757,A -85,B 0,C 180,E1 -22895.037,E2 -22895.037} C_VEL
LIN {X 0,Y 171.352,Z 427.735,A -85,B 0,C 180,E1 -22898.81,E2 -22898.81} C_VEL
LIN {X 0,Y 171.338,Z 427.748,A -85,B 0,C 180,E1 -22904.213,E2 -22904.213} C_VEL
LIN {X 0,Y 171.357,Z 427.754,A -85,B 0,C 180,E1 -22909.59,E2 -22909.59} C_VEL
LIN {X 0,Y 171.507,Z 428.576,A -85,B 0,C 180,E1 -22910.147,E2 -22910.147} C_VEL
LIN {X 0,Y 172.806,Z 431.228,A -85,B 0,C 180,E1 -22910.685,E2 -22910.685} C_VEL
LIN {X 0,Y 174.221,Z 432.708,A -85,B 0,C 180,E1 -22911.185,E2 -22911.185} C_VEL
LIN {X 0,Y 176.193,Z 436.032,A -85,B 0,C 180,E1 -22911.972,E2 -22911.972} C_VEL
LIN {X 0,Y 181.185,Z 444.693,A -85,B 0,C 180,E1 -22914.07,E2 -22914.07} C_VEL
LIN {X 0,Y 185.755,Z 454.239,A -85,B 0,C 180,E1 -22916.344,E2 -22916.344} C_VEL
LIN {X 0,Y 189.688,Z 464.956,A -85,B 0,C 180,E1 -22918.907,E2 -22918.907} C_VEL
LIN {X 0,Y 191.815,Z 473.138,A -85,B 0,C 180,E1 -22920.922,E2 -22920.922} C_VEL
LIN {X 0,Y 189.267,Z 484.374,A -85,B 0,C 180,E1 -22923.006,E2 -22923.006} C_VEL
LIN {X 0,Y 186.306,Z 494.849,A -85,B 0,C 180,E1 -22925.487,E2 -22925.487} C_VEL
LIN {X 0,Y 183.411,Z 503.523,A -85,B 0,C 180,E1 -22928.065,E2 -22928.065} C_VEL
LIN {X 0,Y 180.511,Z 511.952,A -85,B 0,C 180,E1 -22931.267,E2 -22931.267} C_VEL
LIN {X 0,Y 178.313,Z 517.671,A -85,B 0,C 180,E1 -22933.987,E2 -22933.987} C_VEL
LIN {X 0,Y 176.374,Z 523.242,A -85,B 0,C 180,E1 -22937.343,E2 -22937.343} C_VEL
LIN {X 0,Y 174.603,Z 527.644,A -85,B 0,C 180,E1 -22940.737,E2 -22940.737} C_VEL
LIN {X 0,Y 173.651,Z 529.961,A -85,B 0,C 180,E1 -22943.029,E2 -22943.029} C_VEL
LIN {X 0,Y 172.512,Z 533.338,A -85,B 0,C 180,E1 -22947.668,E2 -22947.668} C_VEL
LIN {X 0,Y 172.335,Z 535.025,A -85,B 0,C 180,E1 -22952.34,E2 -22952.34} C_VEL
LIN {X 0,Y 172.328,Z 535.337,A -85,B 0,C 180,E1 -22954.681,E2 -22954.681} C_VEL
LIN {X 0,Y 172.452,Z 535.275,A -85,B 0,C 180,E1 -22957.025,E2 -22957.025} C_VEL
LIN {X 0,Y 174.055,Z 533.817,A -85,B 0,C 180,E1 -22961.65,E2 -22961.65} C_VEL
LIN {X 0,Y 175.156,Z 532.518,A -85,B 0,C 180,E1 -22963.933,E2 -22963.933} C_VEL
LIN {X 0,Y 177.069,Z 529.452,A -85,B 0,C 180,E1 -22967.714,E2 -22967.714} C_VEL
LIN {X 0,Y 179.809,Z 524.562,A -85,B 0,C 180,E1 -22971.799,E2 -22971.799} C_VEL
LIN {X 0,Y 182.466,Z 519.301,A -85,B 0,C 180,E1 -22975.07,E2 -22975.07} C_VEL
LIN {X 0,Y 185.648,Z 512.673,A -85,B 0,C 180,E1 -22978.245,E2 -22978.245} C_VEL
LIN {X 0,Y 189.425,Z 503.979,A -85,B 0,C 180,E1 -22981.422,E2 -22981.422} C_VEL
LIN {X 0,Y 192.642,Z 495.676,A -85,B 0,C 180,E1 -22983.806,E2 -22983.806} C_VEL
LIN {X 0,Y 196.031,Z 485.346,A -85,B 0,C 180,E1 -22986.184,E2 -22986.184} C_VEL
LIN {X 0,Y 196.986,Z 481.874,A -85,B 0,C 180,E1 -22986.868,E2 -22986.868} C_VEL
LIN {X 0,Y 197.002,Z 479.988,A -85,B 0,C 180,E1 -22987.337,E2 -22987.337} C_VEL
LIN {X 0,Y 194.586,Z 470.624,A -85,B 0,C 180,E1 -22990.085,E2 -22990.085} C_VEL
LIN {X 0,Y 191.017,Z 460.741,A -85,B 0,C 180,E1 -22992.933,E2 -22992.933} C_VEL
LIN {X 0,Y 186.581,Z 451.538,A -85,B 0,C 180,E1 -22995.677,E2 -22995.677} C_VEL
LIN {X 0,Y 181.639,Z 443.271,A -85,B 0,C 180,E1 -22998.315,E2 -22998.315} C_VEL
LIN {X 0,Y 175.932,Z 435.28,A -85,B 0,C 180,E1 -23001.139,E2 -23001.139} C_VEL
LIN {X 0,Y 173.304,Z 432.049,A -85,B 0,C 180,E1 -23002.422,E2 -23002.422} C_VEL
LIN {X 0,Y 172.745,Z 431.045,A -85,B 0,C 180,E1 -23002.757,E2 -23002.757} C_VEL
LIN {X 0,Y 171.437,Z 427.755,A -85,B 0,C 180,E1 -23005.702,E2 -23005.702} C_VEL
LIN {X 0,Y 171.483,Z 427.681,A -85,B 0,C 180,E1 -23010.034,E2 -23010.034} C_VEL
LIN {X 0,Y 175.205,Z 442.148,A -85,B 0,C 180,E1 -23012.522,E2 -23012.522} C_VEL
LIN {X 0,Y 178.353,Z 454.753,A -85,B 0,C 180,E1 -23015.005,E2 -23015.005} C_VEL
LIN {X 0,Y 179.093,Z 457.351,A -85,B 0,C 180,E1 -23015.575,E2 -23015.575} C_VEL
LIN {X 0,Y 178.744,Z 461.094,A -85,B 0,C 180,E1 -23016.339,E2 -23016.339} C_VEL
LIN {X 0,Y 176.64,Z 474.064,A -85,B 0,C 180,E1 -23019.322,E2 -23019.322} C_VEL
LIN {X 0,Y 174.943,Z 485.487,A -85,B 0,C 180,E1 -23022.464,E2 -23022.464} C_VEL
LIN {X 0,Y 173.456,Z 496.063,A -85,B 0,C 180,E1 -23025.929,E2 -23025.929} C_VEL
LIN {X 0,Y 172.297,Z 506.556,A -85,B 0,C 180,E1 -23030.016,E2 -23030.016} C_VEL
LIN {X 0,Y 171.363,Z 516.42,A -85,B 0,C 180,E1 -23034.705,E2 -23034.705} C_VEL
LIN {X 0,Y 171.519,Z 523.634,A -85,B 0,C 180,E1 -23038.825,E2 -23038.825} C_VEL
LIN {X 0,Y 172.138,Z 530.43,A -85,B 0,C 180,E1 -23043.511,E2 -23043.511} C_VEL
LIN {X 0,Y 173.715,Z 535.901,A -85,B 0,C 180,E1 -23048.14,E2 -23048.14} C_VEL
LIN {X 0,Y 175.562,Z 539.238,A -85,B 0,C 180,E1 -23051.546,E2 -23051.546} C_VEL
LIN {X 0,Y 179.06,Z 542.643,A -85,B 0,C 180,E1 -23055.946,E2 -23055.946} C_VEL
LIN {X 0,Y 183.524,Z 544.96,A -85,B 0,C 180,E1 -23060.16,E2 -23060.16} C_VEL
LIN {X 0,Y 188.846,Z 546.246,A -85,B 0,C 180,E1 -23064.165,E2 -23064.165} C_VEL
LIN {X 0,Y 195.178,Z 546.512,A -85,B 0,C 180,E1 -23067.911,E2 -23067.911} C_VEL
LIN {X 0,Y 202.461,Z 545.78,A -85,B 0,C 180,E1 -23071.378,E2 -23071.378} C_VEL
LIN {X 0,Y 210.601,Z 544.047,A -85,B 0,C 180,E1 -23074.562,E2 -23074.562} C_VEL
LIN {X 0,Y 219.448,Z 541.344,A -85,B 0,C 180,E1 -23077.48,E2 -23077.48} C_VEL
LIN {X 0,Y 226.54,Z 538.635,A -85,B 0,C 180,E1 -23079.492,E2 -23079.492} C_VEL
LIN {X 0,Y 227.112,Z 538.626,A -85,B 0,C 180,E1 -23080.035,E2 -23080.035} C_VEL
LIN {X 0,Y 220.335,Z 544.083,A -85,B 0,C 180,E1 -23082.806,E2 -23082.806} C_VEL
LIN {X 0,Y 214.083,Z 548.9,A -85,B 0,C 180,E1 -23085.103,E2 -23085.103} C_VEL
LIN {X 0,Y 203.159,Z 556.51,A -85,B 0,C 180,E1 -23088.905,E2 -23088.905} C_VEL
LIN {X 0,Y 197.155,Z 560.57,A -85,B 0,C 180,E1 -23091.402,E2 -23091.402} C_VEL
LIN {X 0,Y 189.508,Z 565.282,A -85,B 0,C 180,E1 -23094.91,E2 -23094.91} C_VEL
LIN {X 0,Y 181.732,Z 570.086,A -85,B 0,C 180,E1 -23099.816,E2 -23099.816} C_VEL
LIN {X 0,Y 176.867,Z 573.023,A -85,B 0,C 180,E1 -23104.079,E2 -23104.079} C_VEL
LIN {X 0,Y 173.282,Z 575.222,A -85,B 0,C 180,E1 -23108.88,E2 -23108.88} C_VEL
LIN {X 0,Y 171.28,Z 576.566,A -85,B 0,C 180,E1 -23114.224,E2 -23114.224} C_VEL
LIN {X 0,Y 170.427,Z 580.205,A -85,B 0,C 180,E1 -23118.098,E2 -23118.098} C_VEL
LIN {X 0,Y 170.438,Z 582.58,A -85,B 0,C 180,E1 -23121.743,E2 -23121.743} C_VEL
LIN {X 0,Y 170.95,Z 583.967,A -85,B 0,C 180,E1 -23125.281,E2 -23125.281} C_VEL
LIN {X 0,Y 171.407,Z 584.384,A -85,B 0,C 180,E1 -23127.648,E2 -23127.648} C_VEL
LIN {X 0,Y 172.084,Z 584.389,A -85,B 0,C 180,E1 -23129.997,E2 -23129.997} C_VEL
LIN {X 0,Y 171.214,Z 583.049,A -85,B 0,C 180,E1 -23133.889,E2 -23133.889} C_VEL
LIN {X 0,Y 170.708,Z 582.396,A -85,B 0,C 180,E1 -23135.177,E2 -23135.177} C_VEL
LIN {X 0,Y 169.116,Z 581.062,A -85,B 0,C 180,E1 -23137.052,E2 -23137.052} C_VEL
LIN {X 0,Y 164.549,Z 576.913,A -85,B 0,C 180,E1 -23141.366,E2 -23141.366} C_VEL
LIN {X 0,Y 163.612,Z 574.749,A -85,B 0,C 180,E1 -23143.28,E2 -23143.28} C_VEL
LIN {X 0,Y 163.603,Z 573.969,A -85,B 0,C 180,E1 -23143.923,E2 -23143.923} C_VEL
LIN {X 0,Y 164.409,Z 569.288,A -85,B 0,C 180,E1 -23147.408,E2 -23147.408} C_VEL
LIN {X 0,Y 166.26,Z 562.106,A -85,B 0,C 180,E1 -23151.571,E2 -23151.571} C_VEL
LIN {X 0,Y 168.784,Z 553.816,A -85,B 0,C 180,E1 -23155.261,E2 -23155.261} C_VEL
LIN {X 0,Y 171.267,Z 545.615,A -85,B 0,C 180,E1 -23158.155,E2 -23158.155} C_VEL
LIN {X 0,Y 172.384,Z 541.87,A -85,B 0,C 180,E1 -23159.287,E2 -23159.287} C_VEL
LIN {X 0,Y 173.493,Z 530.576,A -85,B 0,C 180,E1 -23162.459,E2 -23162.459} C_VEL
LIN {X 0,Y 174.486,Z 519.956,A -85,B 0,C 180,E1 -23164.879,E2 -23164.879} C_VEL
LIN {X 0,Y 175.439,Z 507.315,A -85,B 0,C 180,E1 -23167.174,E2 -23167.174} C_VEL
LIN {X 0,Y 176.101,Z 494.977,A -85,B 0,C 180,E1 -23168.916,E2 -23168.916} C_VEL
LIN {X 0,Y 176.268,Z 484.393,A -85,B 0,C 180,E1 -23170.086,E2 -23170.086} C_VEL
LIN {X 0,Y 174.354,Z 471.274,A -85,B 0,C 180,E1 -23171.596,E2 -23171.596} C_VEL
LIN {X 0,Y 172.121,Z 460.804,A -85,B 0,C 180,E1 -23172.804,E2 -23172.804} C_VEL
LIN {X 0,Y 171.585,Z 453.997,A -85,B 0,C 180,E1 -23174.583,E2 -23174.583} C_VEL
LIN {X 0,Y 170.465,Z 449.847,A -85,B 0,C 180,E1 -23175.933,E2 -23175.933} C_VEL
LIN {X 0,Y 167.891,Z 441.755,A -85,B 0,C 180,E1 -23178.889,E2 -23178.889} C_VEL
LIN {X 0,Y 165.789,Z 434.689,A -85,B 0,C 180,E1 -23181.687,E2 -23181.687} C_VEL
LIN {X 0,Y 164.548,Z 428.608,A -85,B 0,C 180,E1 -23187.124,E2 -23187.124} C_VEL
LIN {X 0,Y 164.385,Z 428.63,A -85,B 0,C 180,E1 -23193.865,E2 -23193.865} C_VEL
LIN {X 0,Y 164.476,Z 428.612,A -85,B 0,C 180,E1 -23200.05,E2 -23200.05} C_VEL
LIN {X 0,Y 164.528,Z 428.606,A -85,B 0,C 180,E1 -23205.15,E2 -23205.15} C_VEL
LIN {X 0,Y 164.789,Z 428.571,A -85,B 0,C 180,E1 -23210.178,E2 -23210.178} C_VEL
LIN {X 0,Y 164.838,Z 428.578,A -85,B 0,C 180,E1 -23212.652,E2 -23212.652} C_VEL
LIN {X 0,Y 165.043,Z 428.552,A -85,B 0,C 180,E1 -23217.56,E2 -23217.56} C_VEL
LIN {X 0,Y 165.289,Z 428.512,A -85,B 0,C 180,E1 -23220.001,E2 -23220.001} C_VEL
LIN {X 0,Y 164.767,Z 428.581,A -85,B 0,C 180,E1 -23224.894,E2 -23224.894} C_VEL
LIN {X 0,Y 164.839,Z 428.539,A -85,B 0,C 180,E1 -23227.349,E2 -23227.349} C_VEL
LIN {X 0,Y 164.743,Z 428.557,A -85,B 0,C 180,E1 -23231.147,E2 -23231.147} C_VEL
LIN {X 0,Y 164.497,Z 428.61,A -85,B 0,C 180,E1 -23237.402,E2 -23237.402} C_VEL
LIN {X 0,Y 164.466,Z 428.624,A -85,B 0,C 180,E1 -23239.991,E2 -23239.991} C_VEL
LIN {X 0,Y 164.386,Z 428.626,A -85,B 0,C 180,E1 -23246.135,E2 -23246.135} C_VEL
LIN {X 0,Y 164.367,Z 428.601,A -85,B 0,C 180,E1 -23251.229,E2 -23251.229} C_VEL
LIN {X 0,Y 164.288,Z 428.618,A -85,B 0,C 180,E1 -23256.792,E2 -23256.792} C_VEL
LIN {X 0,Y 164.287,Z 428.621,A -85,B 0,C 180,E1 -23259.918,E2 -23259.918} C_VEL
LIN {X 0,Y 164.275,Z 428.634,A -85,B 0,C 180,E1 -23263.345,E2 -23263.345} C_VEL
LIN {X 0,Y 164.327,Z 428.764,A -85,B 0,C 180,E1 -23267.292,E2 -23267.292} C_VEL
LIN {X 0,Y 164.612,Z 429.925,A -85,B 0,C 180,E1 -23268,E2 -23268} C_VEL
LIN {X 0,Y 165.988,Z 432.378,A -85,B 0,C 180,E1 -23268.61,E2 -23268.61} C_VEL
LIN {X 0,Y 167.408,Z 434.004,A -85,B 0,C 180,E1 -23269.176,E2 -23269.176} C_VEL
LIN {X 0,Y 169.394,Z 437.192,A -85,B 0,C 180,E1 -23270.039,E2 -23270.039} C_VEL
LIN {X 0,Y 174.124,Z 444.894,A -85,B 0,C 180,E1 -23272.148,E2 -23272.148} C_VEL
LIN {X 0,Y 178.758,Z 454.277,A -85,B 0,C 180,E1 -23274.571,E2 -23274.571} C_VEL
LIN {X 0,Y 182.464,Z 463.792,A -85,B 0,C 180,E1 -23277.007,E2 -23277.007} C_VEL
LIN {X 0,Y 184.879,Z 472.021,A -85,B 0,C 180,E1 -23279.148,E2 -23279.148} C_VEL
LIN {X 0,Y 185.466,Z 474.754,A -85,B 0,C 180,E1 -23279.875,E2 -23279.875} C_VEL
LIN {X 0,Y 184.737,Z 478.964,A -85,B 0,C 180,E1 -23280.675,E2 -23280.675} C_VEL
LIN {X 0,Y 181.922,Z 489.433,A -85,B 0,C 180,E1 -23282.856,E2 -23282.856} C_VEL
LIN {X 0,Y 179.345,Z 497.939,A -85,B 0,C 180,E1 -23285.089,E2 -23285.089} C_VEL
LIN {X 0,Y 176.424,Z 506.253,A -85,B 0,C 180,E1 -23287.766,E2 -23287.766} C_VEL
LIN {X 0,Y 173.4,Z 514.293,A -85,B 0,C 180,E1 -23291.083,E2 -23291.083} C_VEL
LIN {X 0,Y 171.586,Z 518.794,A -85,B 0,C 180,E1 -23293.342,E2 -23293.342} C_VEL
LIN {X 0,Y 169.54,Z 524.336,A -85,B 0,C 180,E1 -23296.824,E2 -23296.824} C_VEL
LIN {X 0,Y 167.676,Z 528.718,A -85,B 0,C 180,E1 -23300.351,E2 -23300.351} C_VEL
LIN {X 0,Y 166.681,Z 531.023,A -85,B 0,C 180,E1 -23302.736,E2 -23302.736} C_VEL
LIN {X 0,Y 165.949,Z 532.907,A -85,B 0,C 180,E1 -23305.144,E2 -23305.144} C_VEL
LIN {X 0,Y 165.492,Z 534.378,A -85,B 0,C 180,E1 -23307.569,E2 -23307.569} C_VEL
LIN {X 0,Y 165.312,Z 536.043,A -85,B 0,C 180,E1 -23312.439,E2 -23312.439} C_VEL
LIN {X 0,Y 165.321,Z 536.346,A -85,B 0,C 180,E1 -23314.88,E2 -23314.88} C_VEL
LIN {X 0,Y 165.472,Z 536.268,A -85,B 0,C 180,E1 -23317.323,E2 -23317.323} C_VEL
LIN {X 0,Y 167.175,Z 534.79,A -85,B 0,C 180,E1 -23322.137,E2 -23322.137} C_VEL
LIN {X 0,Y 168.34,Z 533.482,A -85,B 0,C 180,E1 -23324.509,E2 -23324.509} C_VEL
LIN {X 0,Y 170.389,Z 530.386,A -85,B 0,C 180,E1 -23328.434,E2 -23328.434} C_VEL
LIN {X 0,Y 173.29,Z 525.477,A -85,B 0,C 180,E1 -23332.664,E2 -23332.664} C_VEL
LIN {X 0,Y 176.107,Z 520.194,A -85,B 0,C 180,E1 -23336.041,E2 -23336.041} C_VEL
LIN {X 0,Y 179.473,Z 513.535,A -85,B 0,C 180,E1 -23339.309,E2 -23339.309} C_VEL
LIN {X 0,Y 183.369,Z 504.96,A -85,B 0,C 180,E1 -23342.519,E2 -23342.519} C_VEL
LIN {X 0,Y 186.83,Z 496.458,A -85,B 0,C 180,E1 -23345.008,E2 -23345.008} C_VEL
LIN {X 0,Y 190.21,Z 486.629,A -85,B 0,C 180,E1 -23347.321,E2 -23347.321} C_VEL
LIN {X 0,Y 191.025,Z 483.826,A -85,B 0,C 180,E1 -23347.887,E2 -23347.887} C_VEL
LIN {X 0,Y 190.619,Z 480.768,A -85,B 0,C 180,E1 -23348.815,E2 -23348.815} C_VEL
LIN {X 0,Y 188.227,Z 471.549,A -85,B 0,C 180,E1 -23351.689,E2 -23351.689} C_VEL
LIN {X 0,Y 184.911,Z 462.433,A -85,B 0,C 180,E1 -23354.519,E2 -23354.519} C_VEL
LIN {X 0,Y 180.746,Z 453.828,A -85,B 0,C 180,E1 -23357.33,E2 -23357.33} C_VEL
LIN {X 0,Y 176.063,Z 445.872,A -85,B 0,C 180,E1 -23360.12,E2 -23360.12} C_VEL
LIN {X 0,Y 172.42,Z 440.821,A -85,B 0,C 180,E1 -23362.122,E2 -23362.122} C_VEL
LIN {X 0,Y 169.203,Z 436.586,A -85,B 0,C 180,E1 -23363.892,E2 -23363.892} C_VEL
LIN {X 0,Y 166.338,Z 433.175,A -85,B 0,C 180,E1 -23365.489,E2 -23365.489} C_VEL
LIN {X 0,Y 165.898,Z 432.266,A -85,B 0,C 180,E1 -23365.866,E2 -23365.866} C_VEL
LIN {X 0,Y 164.436,Z 428.63,A -85,B 0,C 180,E1 -23369.675,E2 -23369.675} C_VEL
LIN {X 0,Y 168.515,Z 444.596,A -85,B 0,C 180,E1 -23372.541,E2 -23372.541} C_VEL
LIN {X 0,Y 171.753,Z 457.446,A -85,B 0,C 180,E1 -23375.237,E2 -23375.237} C_VEL
LIN {X 0,Y 172.085,Z 459.026,A -85,B 0,C 180,E1 -23375.592,E2 -23375.592} C_VEL
LIN {X 0,Y 169.974,Z 471.66,A -85,B 0,C 180,E1 -23378.471,E2 -23378.471} C_VEL
LIN {X 0,Y 168.127,Z 483.553,A -85,B 0,C 180,E1 -23381.728,E2 -23381.728} C_VEL
LIN {X 0,Y 166.539,Z 494.571,A -85,B 0,C 180,E1 -23385.332,E2 -23385.332} C_VEL
LIN {X 0,Y 165.293,Z 505.398,A -85,B 0,C 180,E1 -23389.589,E2 -23389.589} C_VEL
LIN {X 0,Y 164.276,Z 515.669,A -85,B 0,C 180,E1 -23394.476,E2 -23394.476} C_VEL
LIN {X 0,Y 164.425,Z 523.193,A -85,B 0,C 180,E1 -23398.775,E2 -23398.775} C_VEL
LIN {X 0,Y 165.05,Z 530.33,A -85,B 0,C 180,E1 -23403.661,E2 -23403.661} C_VEL
LIN {X 0,Y 166.715,Z 536.115,A -85,B 0,C 180,E1 -23408.484,E2 -23408.484} C_VEL
LIN {X 0,Y 168.623,Z 539.633,A -85,B 0,C 180,E1 -23412.028,E2 -23412.028} C_VEL
LIN {X 0,Y 172.279,Z 543.359,A -85,B 0,C 180,E1 -23416.592,E2 -23416.592} C_VEL
LIN {X 0,Y 176.95,Z 546.017,A -85,B 0,C 180,E1 -23420.944,E2 -23420.944} C_VEL
LIN {X 0,Y 182.533,Z 547.661,A -85,B 0,C 180,E1 -23425.057,E2 -23425.057} C_VEL
LIN {X 0,Y 189.141,Z 548.28,A -85,B 0,C 180,E1 -23428.884,E2 -23428.884} C_VEL
LIN {X 0,Y 196.724,Z 547.89,A -85,B 0,C 180,E1 -23432.403,E2 -23432.403} C_VEL
LIN {X 0,Y 205.154,Z 546.533,A -85,B 0,C 180,E1 -23435.617,E2 -23435.617} C_VEL
LIN {X 0,Y 214.302,Z 544.224,A -85,B 0,C 180,E1 -23438.543,E2 -23438.543} C_VEL
LIN {X 0,Y 219.122,Z 542.712,A -85,B 0,C 180,E1 -23439.901,E2 -23439.901} C_VEL
LIN {X 0,Y 217.49,Z 543.994,A -85,B 0,C 180,E1 -23440.705,E2 -23440.705} C_VEL
LIN {X 0,Y 211.328,Z 548.328,A -85,B 0,C 180,E1 -23442.974,E2 -23442.974} C_VEL
LIN {X 0,Y 204.545,Z 552.75,A -85,B 0,C 180,E1 -23445.22,E2 -23445.22} C_VEL
LIN {X 0,Y 195.814,Z 558.193,A -85,B 0,C 180,E1 -23448.393,E2 -23448.393} C_VEL
LIN {X 0,Y 185.579,Z 563.982,A -85,B 0,C 180,E1 -23452.702,E2 -23452.702} C_VEL
LIN {X 0,Y 178.624,Z 567.733,A -85,B 0,C 180,E1 -23456.573,E2 -23456.573} C_VEL
LIN {X 0,Y 172.833,Z 570.767,A -85,B 0,C 180,E1 -23460.791,E2 -23460.791} C_VEL
LIN {X 0,Y 168.518,Z 572.964,A -85,B 0,C 180,E1 -23465.349,E2 -23465.349} C_VEL
LIN {X 0,Y 165.603,Z 574.367,A -85,B 0,C 180,E1 -23470.15,E2 -23470.15} C_VEL
LIN {X 0,Y 164.642,Z 574.948,A -85,B 0,C 180,E1 -23472.932,E2 -23472.932} C_VEL
LIN {X 0,Y 163.398,Z 579.223,A -85,B 0,C 180,E1 -23477.579,E2 -23477.579} C_VEL
LIN {X 0,Y 163.373,Z 581.727,A -85,B 0,C 180,E1 -23481.653,E2 -23481.653} C_VEL
LIN {X 0,Y 163.836,Z 582.958,A -85,B 0,C 180,E1 -23485.076,E2 -23485.076} C_VEL
LIN {X 0,Y 164.322,Z 583.374,A -85,B 0,C 180,E1 -23487.546,E2 -23487.546} C_VEL
LIN {X 0,Y 165.03,Z 583.369,A -85,B 0,C 180,E1 -23489.997,E2 -23489.997} C_VEL
LIN {X 0,Y 164.166,Z 582.162,A -85,B 0,C 180,E1 -23493.7,E2 -23493.7} C_VEL
LIN {X 0,Y 163.619,Z 580.129,A -85,B 0,C 180,E1 -23497.401,E2 -23497.401} C_VEL
LIN {X 0,Y 163.396,Z 576.983,A -85,B 0,C 180,E1 -23501.157,E2 -23501.157} C_VEL
LIN {X 0,Y 163.603,Z 573.969,A -85,B 0,C 180,E1 -23503.923,E2 -23503.923} C_VEL
LIN {X 0,Y 163.284,Z 571.566,A -85,B 0,C 180,E1 -23505.812,E2 -23505.812} C_VEL
LIN {X 0,Y 161.364,Z 567.117,A -85,B 0,C 180,E1 -23508.872,E2 -23508.872} C_VEL
LIN {X 0,Y 159.888,Z 562.107,A -85,B 0,C 180,E1 -23511.88,E2 -23511.88} C_VEL
LIN {X 0,Y 160.26,Z 558.769,A -85,B 0,C 180,E1 -23513.624,E2 -23513.624} C_VEL
LIN {X 0,Y 162.809,Z 551.125,A -85,B 0,C 180,E1 -23516.949,E2 -23516.949} C_VEL
LIN {X 0,Y 165.539,Z 542.599,A -85,B 0,C 180,E1 -23519.92,E2 -23519.92} C_VEL
LIN {X 0,Y 166.845,Z 531.708,A -85,B 0,C 180,E1 -23523.199,E2 -23523.199} C_VEL
LIN {X 0,Y 168.063,Z 520.951,A -85,B 0,C 180,E1 -23525.831,E2 -23525.831} C_VEL
LIN {X 0,Y 169.221,Z 509.212,A -85,B 0,C 180,E1 -23528.15,E2 -23528.15} C_VEL
LIN {X 0,Y 170.166,Z 496.126,A -85,B 0,C 180,E1 -23530.147,E2 -23530.147} C_VEL
LIN {X 0,Y 170.526,Z 485.567,A -85,B 0,C 180,E1 -23531.413,E2 -23531.413} C_VEL
LIN {X 0,Y 168.718,Z 472.237,A -85,B 0,C 180,E1 -23533.097,E2 -23533.097} C_VEL
LIN {X 0,Y 165.984,Z 459.546,A -85,B 0,C 180,E1 -23534.722,E2 -23534.722} C_VEL
LIN {X 0,Y 165.086,Z 454.392,A -85,B 0,C 180,E1 -23536.358,E2 -23536.358} C_VEL
LIN {X 0,Y 162.468,Z 445.932,A -85,B 0,C 180,E1 -23539.545,E2 -23539.545} C_VEL
LIN {X 0,Y 160.335,Z 438.578,A -85,B 0,C 180,E1 -23542.613,E2 -23542.613} C_VEL
LIN {X 0,Y 157.854,Z 431.327,A -85,B 0,C 180,E1 -23546.185,E2 -23546.185} C_VEL
LIN {X 0,Y 157.514,Z 429.484,A -85,B 0,C 180,E1 -23547.059,E2 -23547.059} C_VEL
LIN {X 0,Y 157.315,Z 429.513,A -85,B 0,C 180,E1 -23553.465,E2 -23553.465} C_VEL
LIN {X 0,Y 157.385,Z 429.495,A -85,B 0,C 180,E1 -23559.667,E2 -23559.667} C_VEL
LIN {X 0,Y 157.454,Z 429.486,A -85,B 0,C 180,E1 -23564.467,E2 -23564.467} C_VEL
LIN {X 0,Y 157.718,Z 429.452,A -85,B 0,C 180,E1 -23569.733,E2 -23569.733} C_VEL
LIN {X 0,Y 157.795,Z 429.454,A -85,B 0,C 180,E1 -23572.322,E2 -23572.322} C_VEL
LIN {X 0,Y 158.251,Z 429.389,A -85,B 0,C 180,E1 -23580.001,E2 -23580.001} C_VEL
LIN {X 0,Y 157.777,Z 429.414,A -85,B 0,C 180,E1 -23587.68,E2 -23587.68} C_VEL
LIN {X 0,Y 157.672,Z 429.438,A -85,B 0,C 180,E1 -23591.317,E2 -23591.317} C_VEL
LIN {X 0,Y 157.47,Z 429.492,A -85,B 0,C 180,E1 -23595.533,E2 -23595.533} C_VEL
LIN {X 0,Y 157.363,Z 429.503,A -85,B 0,C 180,E1 -23600.935,E2 -23600.935} C_VEL
LIN {X 0,Y 157.307,Z 429.499,A -85,B 0,C 180,E1 -23606.686,E2 -23606.686} C_VEL
LIN {X 0,Y 157.268,Z 429.498,A -85,B 0,C 180,E1 -23612.43,E2 -23612.43} C_VEL
LIN {X 0,Y 157.262,Z 429.495,A -85,B 0,C 180,E1 -23616.452,E2 -23616.452} C_VEL
LIN {X 0,Y 157.206,Z 429.528,A -85,B 0,C 180,E1 -23622.113,E2 -23622.113} C_VEL
LIN {X 0,Y 157.21,Z 429.639,A -85,B 0,C 180,E1 -23624.499,E2 -23624.499} C_VEL
LIN {X 0,Y 157.643,Z 431.242,A -85,B 0,C 180,E1 -23625.541,E2 -23625.541} C_VEL
LIN {X 0,Y 159.316,Z 433.707,A -85,B 0,C 180,E1 -23626.339,E2 -23626.339} C_VEL
LIN {X 0,Y 160.484,Z 434.869,A -85,B 0,C 180,E1 -23626.85,E2 -23626.85} C_VEL
LIN {X 0,Y 162.457,Z 438.091,A -85,B 0,C 180,E1 -23627.804,E2 -23627.804} C_VEL
LIN {X 0,Y 164.328,Z 440.988,A -85,B 0,C 180,E1 -23628.688,E2 -23628.688} C_VEL
LIN {X 0,Y 168.192,Z 447.341,A -85,B 0,C 180,E1 -23630.628,E2 -23630.628} C_VEL
LIN {X 0,Y 172.564,Z 456.069,A -85,B 0,C 180,E1 -23633.113,E2 -23633.113} C_VEL
LIN {X 0,Y 176.312,Z 465.844,A -85,B 0,C 180,E1 -23635.807,E2 -23635.807} C_VEL
LIN {X 0,Y 178.706,Z 473.972,A -85,B 0,C 180,E1 -23638.083,E2 -23638.083} C_VEL
LIN {X 0,Y 179.33,Z 477.655,A -85,B 0,C 180,E1 -23639.084,E2 -23639.084} C_VEL
LIN {X 0,Y 176.774,Z 487.22,A -85,B 0,C 180,E1 -23641.006,E2 -23641.006} C_VEL
LIN {X 0,Y 173.662,Z 497.264,A -85,B 0,C 180,E1 -23643.569,E2 -23643.569} C_VEL
LIN {X 0,Y 170.509,Z 505.87,A -85,B 0,C 180,E1 -23646.308,E2 -23646.308} C_VEL
LIN {X 0,Y 167.289,Z 514.235,A -85,B 0,C 180,E1 -23649.724,E2 -23649.724} C_VEL
LIN {X 0,Y 164.909,Z 519.911,A -85,B 0,C 180,E1 -23652.646,E2 -23652.646} C_VEL
LIN {X 0,Y 162.721,Z 525.428,A -85,B 0,C 180,E1 -23656.261,E2 -23656.261} C_VEL
LIN {X 0,Y 160.758,Z 529.789,A -85,B 0,C 180,E1 -23659.932,E2 -23659.932} C_VEL
LIN {X 0,Y 159.716,Z 532.085,A -85,B 0,C 180,E1 -23662.417,E2 -23662.417} C_VEL
LIN {X 0,Y 158.951,Z 533.959,A -85,B 0,C 180,E1 -23664.93,E2 -23664.93} C_VEL
LIN {X 0,Y 158.473,Z 535.416,A -85,B 0,C 180,E1 -23667.461,E2 -23667.461} C_VEL
LIN {X 0,Y 158.29,Z 537.06,A -85,B 0,C 180,E1 -23672.547,E2 -23672.547} C_VEL
LIN {X 0,Y 158.316,Z 537.355,A -85,B 0,C 180,E1 -23675.096,E2 -23675.096} C_VEL
LIN {X 0,Y 158.497,Z 537.26,A -85,B 0,C 180,E1 -23677.647,E2 -23677.647} C_VEL
LIN {X 0,Y 160.309,Z 535.763,A -85,B 0,C 180,E1 -23682.665,E2 -23682.665} C_VEL
LIN {X 0,Y 161.542,Z 534.445,A -85,B 0,C 180,E1 -23685.134,E2 -23685.134} C_VEL
LIN {X 0,Y 163.738,Z 531.319,A -85,B 0,C 180,E1 -23689.213,E2 -23689.213} C_VEL
LIN {X 0,Y 166.816,Z 526.392,A -85,B 0,C 180,E1 -23693.596,E2 -23693.596} C_VEL
LIN {X 0,Y 169.809,Z 521.086,A -85,B 0,C 180,E1 -23697.084,E2 -23697.084} C_VEL
LIN {X 0,Y 173.365,Z 514.394,A -85,B 0,C 180,E1 -23700.449,E2 -23700.449} C_VEL
LIN {X 0,Y 177.384,Z 505.941,A -85,B 0,C 180,E1 -23703.691,E2 -23703.691} C_VEL
LIN {X 0,Y 181.108,Z 497.24,A -85,B 0,C 180,E1 -23706.286,E2 -23706.286} C_VEL
LIN {X 0,Y 184.765,Z 486.896,A -85,B 0,C 180,E1 -23708.748,E2 -23708.748} C_VEL
LIN {X 0,Y 185.105,Z 485.815,A -85,B 0,C 180,E1 -23708.967,E2 -23708.967} C_VEL
LIN {X 0,Y 183.455,Z 477.71,A -85,B 0,C 180,E1 -23711.686,E2 -23711.686} C_VEL
LIN {X 0,Y 180.664,Z 468.704,A -85,B 0,C 180,E1 -23714.691,E2 -23714.691} C_VEL
LIN {X 0,Y 176.568,Z 459.141,A -85,B 0,C 180,E1 -23718.003,E2 -23718.003} C_VEL
LIN {X 0,Y 171.53,Z 450.205,A -85,B 0,C 180,E1 -23721.411,E2 -23721.411} C_VEL
LIN {X 0,Y 168.53,Z 445.918,A -85,B 0,C 180,E1 -23723.284,E2 -23723.284} C_VEL
LIN {X 0,Y 166.091,Z 442.44,A -85,B 0,C 180,E1 -23724.826,E2 -23724.826} C_VEL
LIN {X 0,Y 162.489,Z 437.835,A -85,B 0,C 180,E1 -23727.087,E2 -23727.087} C_VEL
LIN {X 0,Y 159.305,Z 434.408,A -85,B 0,C 180,E1 -23729.145,E2 -23729.145} C_VEL
LIN {X 0,Y 158.367,Z 433.664,A -85,B 0,C 180,E1 -23730.003,E2 -23730.003} C_VEL
LIN {X 0,Y 162.471,Z 449.583,A -85,B 0,C 180,E1 -23733.152,E2 -23733.152} C_VEL
LIN {X 0,Y 164.908,Z 459.864,A -85,B 0,C 180,E1 -23735.447,E2 -23735.447} C_VEL
LIN {X 0,Y 162.539,Z 473.73,A -85,B 0,C 180,E1 -23738.768,E2 -23738.768} C_VEL
LIN {X 0,Y 160.741,Z 485.411,A -85,B 0,C 180,E1 -23742.178,E2 -23742.178} C_VEL
LIN {X 0,Y 159.151,Z 496.591,A -85,B 0,C 180,E1 -23746.073,E2 -23746.073} C_VEL
LIN {X 0,Y 157.98,Z 506.959,A -85,B 0,C 180,E1 -23750.396,E2 -23750.396} C_VEL
LIN {X 0,Y 157.202,Z 515.961,A -85,B 0,C 180,E1 -23754.869,E2 -23754.869} C_VEL
LIN {X 0,Y 157.336,Z 522.621,A -85,B 0,C 180,E1 -23758.72,E2 -23758.72} C_VEL
LIN {X 0,Y 157.969,Z 530.062,A -85,B 0,C 180,E1 -23763.826,E2 -23763.826} C_VEL
LIN {X 0,Y 159.723,Z 536.156,A -85,B 0,C 180,E1 -23768.858,E2 -23768.858} C_VEL
LIN {X 0,Y 162.552,Z 541.045,A -85,B 0,C 180,E1 -23773.756,E2 -23773.756} C_VEL
LIN {X 0,Y 165.514,Z 543.983,A -85,B 0,C 180,E1 -23777.291,E2 -23777.291} C_VEL
LIN {X 0,Y 170.408,Z 546.95,A -85,B 0,C 180,E1 -23781.788,E2 -23781.788} C_VEL
LIN {X 0,Y 176.238,Z 548.916,A -85,B 0,C 180,E1 -23786.018,E2 -23786.018} C_VEL
LIN {X 0,Y 183.124,Z 549.892,A -85,B 0,C 180,E1 -23789.928,E2 -23789.928} C_VEL
LIN {X 0,Y 191.011,Z 549.894,A -85,B 0,C 180,E1 -23793.497,E2 -23793.497} C_VEL
LIN {X 0,Y 199.75,Z 548.95,A -85,B 0,C 180,E1 -23796.735,E2 -23796.735} C_VEL
LIN {X 0,Y 210.092,Z 546.831,A -85,B 0,C 180,E1 -23799.911,E2 -23799.911} C_VEL
LIN {X 0,Y 209.6,Z 547.384,A -85,B 0,C 180,E1 -23800.477,E2 -23800.477} C_VEL
LIN {X 0,Y 201.993,Z 552.016,A -85,B 0,C 180,E1 -23803.056,E2 -23803.056} C_VEL
LIN {X 0,Y 190.538,Z 558.332,A -85,B 0,C 180,E1 -23806.968,E2 -23806.968} C_VEL
LIN {X 0,Y 179.595,Z 563.802,A -85,B 0,C 180,E1 -23811.503,E2 -23811.503} C_VEL
LIN {X 0,Y 172.723,Z 567.059,A -85,B 0,C 180,E1 -23815.271,E2 -23815.271} C_VEL
LIN {X 0,Y 166.667,Z 569.728,A -85,B 0,C 180,E1 -23819.599,E2 -23819.599} C_VEL
LIN {X 0,Y 162.095,Z 571.661,A -85,B 0,C 180,E1 -23824.303,E2 -23824.303} C_VEL
LIN {X 0,Y 158.465,Z 572.961,A -85,B 0,C 180,E1 -23830.569,E2 -23830.569} C_VEL
LIN {X 0,Y 158.146,Z 573.141,A -85,B 0,C 180,E1 -23831.37,E2 -23831.37} C_VEL
LIN {X 0,Y 156.667,Z 577.267,A -85,B 0,C 180,E1 -23835.713,E2 -23835.713} C_VEL
LIN {X 0,Y 156.22,Z 579.907,A -85,B 0,C 180,E1 -23839.63,E2 -23839.63} C_VEL
LIN {X 0,Y 156.364,Z 581.129,A -85,B 0,C 180,E1 -23842.248,E2 -23842.248} C_VEL
LIN {X 0,Y 156.731,Z 581.951,A -85,B 0,C 180,E1 -23844.852,E2 -23844.852} C_VEL
LIN {X 0,Y 157.231,Z 582.364,A -85,B 0,C 180,E1 -23847.435,E2 -23847.435} C_VEL
LIN {X 0,Y 157.974,Z 582.349,A -85,B 0,C 180,E1 -23849.997,E2 -23849.997} C_VEL
LIN {X 0,Y 157.333,Z 581.672,A -85,B 0,C 180,E1 -23852.557,E2 -23852.557} C_VEL
LIN {X 0,Y 156.881,Z 580.587,A -85,B 0,C 180,E1 -23855.138,E2 -23855.138} C_VEL
LIN {X 0,Y 156.449,Z 578.303,A -85,B 0,C 180,E1 -23858.781,E2 -23858.781} C_VEL
LIN {X 0,Y 156.418,Z 574.586,A -85,B 0,C 180,E1 -23862.98,E2 -23862.98} C_VEL
LIN {X 0,Y 157.125,Z 569.971,A -85,B 0,C 180,E1 -23866.899,E2 -23866.899} C_VEL
LIN {X 0,Y 158.617,Z 564.147,A -85,B 0,C 180,E1 -23870.757,E2 -23870.757} C_VEL
LIN {X 0,Y 160.26,Z 558.769,A -85,B 0,C 180,E1 -23873.624,E2 -23873.624} C_VEL
LIN {X 0,Y 160.798,Z 555.258,A -85,B 0,C 180,E1 -23875.31,E2 -23875.31} C_VEL
LIN {X 0,Y 160.141,Z 549.146,A -85,B 0,C 180,E1 -23878.085,E2 -23878.085} C_VEL
LIN {X 0,Y 159.236,Z 541.221,A -85,B 0,C 180,E1 -23881.291,E2 -23881.291} C_VEL
LIN {X 0,Y 159.455,Z 538.309,A -85,B 0,C 180,E1 -23882.286,E2 -23882.286} C_VEL
LIN {X 0,Y 160.865,Z 527.918,A -85,B 0,C 180,E1 -23885.368,E2 -23885.368} C_VEL
LIN {X 0,Y 162.389,Z 516.217,A -85,B 0,C 180,E1 -23888.136,E2 -23888.136} C_VEL
LIN {X 0,Y 163.691,Z 504.64,A -85,B 0,C 180,E1 -23890.307,E2 -23890.307} C_VEL
LIN {X 0,Y 164.714,Z 491.856,A -85,B 0,C 180,E1 -23892.183,E2 -23892.183} C_VEL
LIN {X 0,Y 164.761,Z 486.078,A -85,B 0,C 180,E1 -23892.938,E2 -23892.938} C_VEL
LIN {X 0,Y 163.134,Z 472.664,A -85,B 0,C 180,E1 -23894.761,E2 -23894.761} C_VEL
LIN {X 0,Y 160.802,Z 462.05,A -85,B 0,C 180,E1 -23896.225,E2 -23896.225} C_VEL
LIN {X 0,Y 159.48,Z 458.562,A -85,B 0,C 180,E1 -23896.918,E2 -23896.918} C_VEL
LIN {X 0,Y 156.645,Z 448.997,A -85,B 0,C 180,E1 -23900.716,E2 -23900.716} C_VEL
LIN {X 0,Y 154.747,Z 442.055,A -85,B 0,C 180,E1 -23903.815,E2 -23903.815} C_VEL
LIN {X 0,Y 152.659,Z 435.27,A -85,B 0,C 180,E1 -23907.221,E2 -23907.221} C_VEL
LIN {X 0,Y 150.537,Z 431.613,A -85,B 0,C 180,E1 -23909.876,E2 -23909.876} C_VEL
LIN {X 0,Y 150.26,Z 430.384,A -85,B 0,C 180,E1 -23910.587,E2 -23910.587} C_VEL
LIN {X 0,Y 150.218,Z 430.389,A -85,B 0,C 180,E1 -23915.099,E2 -23915.099} C_VEL
LIN {X 0,Y 150.353,Z 430.374,A -85,B 0,C 180,E1 -23920.901,E2 -23920.901} C_VEL
LIN {X 0,Y 150.443,Z 430.367,A -85,B 0,C 180,E1 -23926.493,E2 -23926.493} C_VEL
LIN {X 0,Y 150.644,Z 430.334,A -85,B 0,C 180,E1 -23929.246,E2 -23929.246} C_VEL
LIN {X 0,Y 150.731,Z 430.333,A -85,B 0,C 180,E1 -23931.96,E2 -23931.96} C_VEL
LIN {X 0,Y 151.212,Z 430.265,A -85,B 0,C 180,E1 -23940.001,E2 -23940.001} C_VEL
LIN {X 0,Y 150.716,Z 430.289,A -85,B 0,C 180,E1 -23948.042,E2 -23948.042} C_VEL
LIN {X 0,Y 150.603,Z 430.318,A -85,B 0,C 180,E1 -23951.502,E2 -23951.502} C_VEL
LIN {X 0,Y 150.374,Z 430.37,A -85,B 0,C 180,E1 -23956.286,E2 -23956.286} C_VEL
LIN {X 0,Y 150.344,Z 430.378,A -85,B 0,C 180,E1 -23960.794,E2 -23960.794} C_VEL
LIN {X 0,Y 150.237,Z 430.367,A -85,B 0,C 180,E1 -23967.284,E2 -23967.284} C_VEL
LIN {X 0,Y 150.208,Z 430.379,A -85,B 0,C 180,E1 -23972.634,E2 -23972.634} C_VEL
LIN {X 0,Y 150.167,Z 430.37,A -85,B 0,C 180,E1 -23977.476,E2 -23977.476} C_VEL
LIN {X 0,Y 150.192,Z 430.566,A -85,B 0,C 180,E1 -23981.275,E2 -23981.275} C_VEL
LIN {X 0,Y 150.708,Z 432.388,A -85,B 0,C 180,E1 -23982.722,E2 -23982.722} C_VEL
LIN {X 0,Y 152.315,Z 434.675,A -85,B 0,C 180,E1 -23983.593,E2 -23983.593} C_VEL
LIN {X 0,Y 153.901,Z 436.538,A -85,B 0,C 180,E1 -23984.4,E2 -23984.4} C_VEL
LIN {X 0,Y 156.138,Z 439.696,A -85,B 0,C 180,E1 -23985.575,E2 -23985.575} C_VEL
LIN {X 0,Y 160.073,Z 445.895,A -85,B 0,C 180,E1 -23987.692,E2 -23987.692} C_VEL
LIN {X 0,Y 164.578,Z 453.933,A -85,B 0,C 180,E1 -23990.32,E2 -23990.32} C_VEL
LIN {X 0,Y 168.799,Z 463.68,A -85,B 0,C 180,E1 -23993.274,E2 -23993.274} C_VEL
LIN {X 0,Y 172.055,Z 473.874,A -85,B 0,C 180,E1 -23996.318,E2 -23996.318} C_VEL
LIN {X 0,Y 173.185,Z 478.86,A -85,B 0,C 180,E1 -23997.821,E2 -23997.821} C_VEL
LIN {X 0,Y 171.986,Z 484.219,A -85,B 0,C 180,E1 -23998.946,E2 -23998.946} C_VEL
LIN {X 0,Y 168.783,Z 494.448,A -85,B 0,C 180,E1 -24001.366,E2 -24001.366} C_VEL
LIN {X 0,Y 165.395,Z 503.834,A -85,B 0,C 180,E1 -24004.183,E2 -24004.183} C_VEL
LIN {X 0,Y 162.345,Z 511.453,A -85,B 0,C 180,E1 -24007.073,E2 -24007.073} C_VEL
LIN {X 0,Y 159.219,Z 518.87,A -85,B 0,C 180,E1 -24010.67,E2 -24010.67} C_VEL
LIN {X 0,Y 156.671,Z 524.8,A -85,B 0,C 180,E1 -24014.389,E2 -24014.389} C_VEL
LIN {X 0,Y 154.508,Z 529.514,A -85,B 0,C 180,E1 -24018.192,E2 -24018.192} C_VEL
LIN {X 0,Y 152.756,Z 533.147,A -85,B 0,C 180,E1 -24022.069,E2 -24022.069} C_VEL
LIN {X 0,Y 151.955,Z 535.012,A -85,B 0,C 180,E1 -24024.695,E2 -24024.695} C_VEL
LIN {X 0,Y 151.455,Z 536.453,A -85,B 0,C 180,E1 -24027.343,E2 -24027.343} C_VEL
LIN {X 0,Y 151.268,Z 538.078,A -85,B 0,C 180,E1 -24032.666,E2 -24032.666} C_VEL
LIN {X 0,Y 151.313,Z 538.364,A -85,B 0,C 180,E1 -24035.333,E2 -24035.333} C_VEL
LIN {X 0,Y 151.527,Z 538.252,A -85,B 0,C 180,E1 -24038.001,E2 -24038.001} C_VEL
LIN {X 0,Y 153.458,Z 536.736,A -85,B 0,C 180,E1 -24043.24,E2 -24043.24} C_VEL
LIN {X 0,Y 154.764,Z 535.406,A -85,B 0,C 180,E1 -24045.814,E2 -24045.814} C_VEL
LIN {X 0,Y 157.095,Z 532.278,A -85,B 0,C 180,E1 -24050.033,E2 -24050.033} C_VEL
LIN {X 0,Y 160.391,Z 527.307,A -85,B 0,C 180,E1 -24054.602,E2 -24054.602} C_VEL
LIN {X 0,Y 163.567,Z 521.978,A -85,B 0,C 180,E1 -24058.208,E2 -24058.208} C_VEL
LIN {X 0,Y 167.327,Z 515.25,A -85,B 0,C 180,E1 -24061.672,E2 -24061.672} C_VEL
LIN {X 0,Y 171.559,Z 506.763,A -85,B 0,C 180,E1 -24064.998,E2 -24064.998} C_VEL
LIN {X 0,Y 175.472,Z 498.024,A -85,B 0,C 180,E1 -24067.649,E2 -24067.649} C_VEL
LIN {X 0,Y 178.756,Z 489.263,A -85,B 0,C 180,E1 -24069.803,E2 -24069.803} C_VEL
LIN {X 0,Y 179.101,Z 487.846,A -85,B 0,C 180,E1 -24070.153,E2 -24070.153} C_VEL
LIN {X 0,Y 177.487,Z 479.588,A -85,B 0,C 180,E1 -24073.124,E2 -24073.124} C_VEL
LIN {X 0,Y 174.732,Z 470.526,A -85,B 0,C 180,E1 -24076.388,E2 -24076.388} C_VEL
LIN {X 0,Y 171.191,Z 462.159,A -85,B 0,C 180,E1 -24079.568,E2 -24079.568} C_VEL
LIN {X 0,Y 167.169,Z 454.772,A -85,B 0,C 180,E1 -24082.652,E2 -24082.652} C_VEL
LIN {X 0,Y 162.922,Z 448.338,A -85,B 0,C 180,E1 -24085.702,E2 -24085.702} C_VEL
LIN {X 0,Y 159.58,Z 443.766,A -85,B 0,C 180,E1 -24088.096,E2 -24088.096} C_VEL
LIN {X 0,Y 157.746,Z 443.651,A -85,B 0,C 180,E1 -24089.178,E2 -24089.178} C_VEL
LIN {X 0,Y 155.928,Z 445.435,A -85,B 0,C 180,E1 -24090.091,E2 -24090.091} C_VEL
LIN {X 0,Y 154.333,Z 445.389,A -85,B 0,C 180,E1 -24091.125,E2 -24091.125} C_VEL
LIN {X 0,Y 153.794,Z 444.378,A -85,B 0,C 180,E1 -24091.645,E2 -24091.645} C_VEL
LIN {X 0,Y 157.047,Z 457.05,A -85,B 0,C 180,E1 -24094.449,E2 -24094.449} C_VEL
LIN {X 0,Y 157.679,Z 460.955,A -85,B 0,C 180,E1 -24095.379,E2 -24095.379} C_VEL
LIN {X 0,Y 155.321,Z 474.465,A -85,B 0,C 180,E1 -24098.777,E2 -24098.777} C_VEL
LIN {X 0,Y 153.378,Z 487.128,A -85,B 0,C 180,E1 -24102.671,E2 -24102.671} C_VEL
LIN {X 0,Y 151.845,Z 497.843,A -85,B 0,C 180,E1 -24106.619,E2 -24106.619} C_VEL
LIN {X 0,Y 150.838,Z 507.042,A -85,B 0,C 180,E1 -24110.614,E2 -24110.614} C_VEL
LIN {X 0,Y 150.101,Z 516.182,A -85,B 0,C 180,E1 -24115.299,E2 -24115.299} C_VEL
LIN {X 0,Y 150.356,Z 523.979,A -85,B 0,C 180,E1 -24119.999,E2 -24119.999} C_VEL
LIN {X 0,Y 151.222,Z 531.394,A -85,B 0,C 180,E1 -24125.333,E2 -24125.333} C_VEL
LIN {X 0,Y 153.254,Z 537.497,A -85,B 0,C 180,E1 -24130.569,E2 -24130.569} C_VEL
LIN {X 0,Y 156.619,Z 542.422,A -85,B 0,C 180,E1 -24135.618,E2 -24135.618} C_VEL
LIN {X 0,Y 161.157,Z 546.264,A -85,B 0,C 180,E1 -24140.418,E2 -24140.418} C_VEL
LIN {X 0,Y 166.828,Z 549.079,A -85,B 0,C 180,E1 -24144.914,E2 -24144.914} C_VEL
LIN {X 0,Y 173.471,Z 550.881,A -85,B 0,C 180,E1 -24149.088,E2 -24149.088} C_VEL
LIN {X 0,Y 181.163,Z 551.705,A -85,B 0,C 180,E1 -24152.895,E2 -24152.895} C_VEL
LIN {X 0,Y 189.737,Z 551.611,A -85,B 0,C 180,E1 -24156.345,E2 -24156.345} C_VEL
LIN {X 0,Y 200.555,Z 550.354,A -85,B 0,C 180,E1 -24159.841,E2 -24159.841} C_VEL
LIN {X 0,Y 199.345,Z 551.403,A -85,B 0,C 180,E1 -24160.882,E2 -24160.882} C_VEL
LIN {X 0,Y 185.399,Z 558.336,A -85,B 0,C 180,E1 -24165.467,E2 -24165.467} C_VEL
LIN {X 0,Y 173.6,Z 563.521,A -85,B 0,C 180,E1 -24170.281,E2 -24170.281} C_VEL
LIN {X 0,Y 166.927,Z 566.259,A -85,B 0,C 180,E1 -24173.881,E2 -24173.881} C_VEL
LIN {X 0,Y 157.968,Z 569.522,A -85,B 0,C 180,E1 -24180.697,E2 -24180.697} C_VEL
LIN {X 0,Y 153.483,Z 570.864,A -85,B 0,C 180,E1 -24186.319,E2 -24186.319} C_VEL
LIN {X 0,Y 151.823,Z 571.259,A -85,B 0,C 180,E1 -24189.682,E2 -24189.682} C_VEL
LIN {X 0,Y 150.091,Z 575.188,A -85,B 0,C 180,E1 -24193.68,E2 -24193.68} C_VEL
LIN {X 0,Y 149.459,Z 577.268,A -85,B 0,C 180,E1 -24196.399,E2 -24196.399} C_VEL
LIN {X 0,Y 149.253,Z 579.966,A -85,B 0,C 180,E1 -24201.432,E2 -24201.432} C_VEL
LIN {X 0,Y 149.632,Z 580.944,A -85,B 0,C 180,E1 -24204.607,E2 -24204.607} C_VEL
LIN {X 0,Y 150.136,Z 581.353,A -85,B 0,C 180,E1 -24207.314,E2 -24207.314} C_VEL
LIN {X 0,Y 150.916,Z 581.328,A -85,B 0,C 180,E1 -24209.997,E2 -24209.997} C_VEL
LIN {X 0,Y 150.236,Z 580.637,A -85,B 0,C 180,E1 -24212.678,E2 -24212.678} C_VEL
LIN {X 0,Y 149.777,Z 579.54,A -85,B 0,C 180,E1 -24215.382,E2 -24215.382} C_VEL
LIN {X 0,Y 149.372,Z 577.47,A -85,B 0,C 180,E1 -24218.867,E2 -24218.867} C_VEL
LIN {X 0,Y 149.4,Z 573.494,A -85,B 0,C 180,E1 -24223.601,E2 -24223.601} C_VEL
LIN {X 0,Y 150.253,Z 568.863,A -85,B 0,C 180,E1 -24227.697,E2 -24227.697} C_VEL
LIN {X 0,Y 151.896,Z 563.016,A -85,B 0,C 180,E1 -24231.721,E2 -24231.721} C_VEL
LIN {X 0,Y 154.359,Z 555.743,A -85,B 0,C 180,E1 -24235.625,E2 -24235.625} C_VEL
LIN {X 0,Y 157.494,Z 546.696,A -85,B 0,C 180,E1 -24239.394,E2 -24239.394} C_VEL
LIN {X 0,Y 158.719,Z 543.209,A -85,B 0,C 180,E1 -24240.608,E2 -24240.608} C_VEL
LIN {X 0,Y 159.455,Z 538.309,A -85,B 0,C 180,E1 -24242.286,E2 -24242.286} C_VEL
LIN {X 0,Y 159.485,Z 534.033,A -85,B 0,C 180,E1 -24243.753,E2 -24243.753} C_VEL
LIN {X 0,Y 157.935,Z 527.071,A -85,B 0,C 180,E1 -24246.244,E2 -24246.244} C_VEL
LIN {X 0,Y 156.435,Z 519.729,A -85,B 0,C 180,E1 -24248.612,E2 -24248.612} C_VEL
LIN {X 0,Y 156.504,Z 514.859,A -85,B 0,C 180,E1 -24249.836,E2 -24249.836} C_VEL
LIN {X 0,Y 158.128,Z 502.326,A -85,B 0,C 180,E1 -24252.217,E2 -24252.217} C_VEL
LIN {X 0,Y 159.224,Z 490.666,A -85,B 0,C 180,E1 -24253.934,E2 -24253.934} C_VEL
LIN {X 0,Y 158.514,Z 479.526,A -85,B 0,C 180,E1 -24255.62,E2 -24255.62} C_VEL
LIN {X 0,Y 156.5,Z 467.024,A -85,B 0,C 180,E1 -24257.436,E2 -24257.436} C_VEL
LIN {X 0,Y 155.01,Z 462.706,A -85,B 0,C 180,E1 -24258.277,E2 -24258.277} C_VEL
LIN {X 0,Y 152.333,Z 457.158,A -85,B 0,C 180,E1 -24259.767,E2 -24259.767} C_VEL
LIN {X 0,Y 149.606,Z 446.679,A -85,B 0,C 180,E1 -24264.397,E2 -24264.397} C_VEL
LIN {X 0,Y 147.38,Z 439.301,A -85,B 0,C 180,E1 -24268.363,E2 -24268.363} C_VEL
LIN {X 0,Y 145.91,Z 437.063,A -85,B 0,C 180,E1 -24270.105,E2 -24270.105} C_VEL
LIN {X 0,Y 145.402,Z 435.586,A -85,B 0,C 180,E1 -24271.096,E2 -24271.096} C_VEL
LIN {X 0,Y 143.449,Z 432.546,A -85,B 0,C 180,E1 -24273.837,E2 -24273.837} C_VEL
LIN {X 0,Y 143.178,Z 431.266,A -85,B 0,C 180,E1 -24274.759,E2 -24274.759} C_VEL
LIN {X 0,Y 143.299,Z 431.249,A -85,B 0,C 180,E1 -24279.922,E2 -24279.922} C_VEL
LIN {X 0,Y 143.361,Z 431.244,A -85,B 0,C 180,E1 -24285.812,E2 -24285.812} C_VEL
LIN {X 0,Y 143.586,Z 431.216,A -85,B 0,C 180,E1 -24288.71,E2 -24288.71} C_VEL
LIN {X 0,Y 143.652,Z 431.21,A -85,B 0,C 180,E1 -24291.561,E2 -24291.561} C_VEL
LIN {X 0,Y 144.17,Z 431.142,A -85,B 0,C 180,E1 -24300.001,E2 -24300.001} C_VEL
LIN {X 0,Y 143.64,Z 431.167,A -85,B 0,C 180,E1 -24308.441,E2 -24308.441} C_VEL
LIN {X 0,Y 143.54,Z 431.198,A -85,B 0,C 180,E1 -24311.714,E2 -24311.714} C_VEL
LIN {X 0,Y 143.308,Z 431.247,A -85,B 0,C 180,E1 -24317.113,E2 -24317.113} C_VEL
LIN {X 0,Y 143.27,Z 431.255,A -85,B 0,C 180,E1 -24321.256,E2 -24321.256} C_VEL
LIN {X 0,Y 143.183,Z 431.237,A -85,B 0,C 180,E1 -24327.939,E2 -24327.939} C_VEL
LIN {X 0,Y 143.158,Z 431.269,A -85,B 0,C 180,E1 -24333.435,E2 -24333.435} C_VEL
LIN {X 0,Y 143.138,Z 431.263,A -85,B 0,C 180,E1 -24337.24,E2 -24337.24} C_VEL
LIN {X 0,Y 143.797,Z 433.61,A -85,B 0,C 180,E1 -24339.448,E2 -24339.448} C_VEL
LIN {X 0,Y 145.594,Z 435.854,A -85,B 0,C 180,E1 -24340.554,E2 -24340.554} C_VEL
LIN {X 0,Y 147.662,Z 438.593,A -85,B 0,C 180,E1 -24341.786,E2 -24341.786} C_VEL
LIN {X 0,Y 150.228,Z 441.905,A -85,B 0,C 180,E1 -24343.288,E2 -24343.288} C_VEL
LIN {X 0,Y 153.561,Z 447.108,A -85,B 0,C 180,E1 -24345.302,E2 -24345.302} C_VEL
LIN {X 0,Y 158.003,Z 454.915,A -85,B 0,C 180,E1 -24348.153,E2 -24348.153} C_VEL
LIN {X 0,Y 162.188,Z 464.139,A -85,B 0,C 180,E1 -24351.26,E2 -24351.26} C_VEL
LIN {X 0,Y 165.047,Z 472.668,A -85,B 0,C 180,E1 -24354.005,E2 -24354.005} C_VEL
LIN {X 0,Y 167.16,Z 481.485,A -85,B 0,C 180,E1 -24356.872,E2 -24356.872} C_VEL
LIN {X 0,Y 163.671,Z 492.713,A -85,B 0,C 180,E1 -24359.382,E2 -24359.382} C_VEL
LIN {X 0,Y 160.529,Z 501.561,A -85,B 0,C 180,E1 -24361.928,E2 -24361.928} C_VEL
LIN {X 0,Y 157.176,Z 509.741,A -85,B 0,C 180,E1 -24364.866,E2 -24364.866} C_VEL
LIN {X 0,Y 153.655,Z 517.696,A -85,B 0,C 180,E1 -24368.54,E2 -24368.54} C_VEL
LIN {X 0,Y 150.797,Z 524.078,A -85,B 0,C 180,E1 -24372.369,E2 -24372.369} C_VEL
LIN {X 0,Y 148.35,Z 529.173,A -85,B 0,C 180,E1 -24376.301,E2 -24376.301} C_VEL
LIN {X 0,Y 146.437,Z 533.122,A -85,B 0,C 180,E1 -24380.333,E2 -24380.333} C_VEL
LIN {X 0,Y 144.963,Z 536.065,A -85,B 0,C 180,E1 -24384.439,E2 -24384.439} C_VEL
LIN {X 0,Y 144.436,Z 537.488,A -85,B 0,C 180,E1 -24387.214,E2 -24387.214} C_VEL
LIN {X 0,Y 144.246,Z 539.096,A -85,B 0,C 180,E1 -24392.796,E2 -24392.796} C_VEL
LIN {X 0,Y 144.314,Z 539.373,A -85,B 0,C 180,E1 -24395.592,E2 -24395.592} C_VEL
LIN {X 0,Y 144.564,Z 539.244,A -85,B 0,C 180,E1 -24398.389,E2 -24398.389} C_VEL
LIN {X 0,Y 146.623,Z 537.709,A -85,B 0,C 180,E1 -24403.869,E2 -24403.869} C_VEL
LIN {X 0,Y 148.011,Z 536.366,A -85,B 0,C 180,E1 -24406.556,E2 -24406.556} C_VEL
LIN {X 0,Y 150.453,Z 533.271,A -85,B 0,C 180,E1 -24410.891,E2 -24410.891} C_VEL
LIN {X 0,Y 154.019,Z 528.222,A -85,B 0,C 180,E1 -24415.692,E2 -24415.692} C_VEL
LIN {X 0,Y 157.392,Z 522.871,A -85,B 0,C 180,E1 -24419.421,E2 -24419.421} C_VEL
LIN {X 0,Y 161.37,Z 516.105,A -85,B 0,C 180,E1 -24422.987,E2 -24422.987} C_VEL
LIN {X 0,Y 165.831,Z 507.585,A -85,B 0,C 180,E1 -24426.396,E2 -24426.396} C_VEL
LIN {X 0,Y 169.938,Z 498.81,A -85,B 0,C 180,E1 -24429.103,E2 -24429.103} C_VEL
LIN {X 0,Y 172.925,Z 491.227,A -85,B 0,C 180,E1 -24431.015,E2 -24431.015} C_VEL
LIN {X 0,Y 173.14,Z 489.938,A -85,B 0,C 180,E1 -24431.405,E2 -24431.405} C_VEL
